FUNCTION_BLOCK "FB_MFC_Sort_COY_Result"
{ S7_Optimized_Access := 'TRUE' }
VERSION : 0.1
// ATTRIBUTES
// AUTO_NUMBER = True
// BLOCK_NUMBER = 117
// END_ATTRIBUTES
   VAR_INPUT
      ii_GINRangeStart { ExternalAccessible := 'False'; ExternalVisible := 'False'; ExternalWritable := 'False'} : Int := 0;   // GIN range start value
      ii_GINRangeEnd { ExternalAccessible := 'False'; ExternalVisible := 'False'; ExternalWritable := 'False'} : Int := 0;   // GIN range end value
      is_ObjectID : String[10];   // Recived parcel identifier
      ii_SourceNode : Int;   // ID Source Node
      ii_DestinationNode : Int;   // ID Destination Node
   END_VAR

   VAR_OUTPUT
      qx_Error : Bool;   // TRUE when collective block error occurred
      qx_Warning : Bool;   // TRUE when collective block warning occurred
   END_VAR

   VAR_IN_OUT
      iq_UDT_FifoHeader : "UDT_FifoHeader";   // FIFO header
      iqa_FifoData : Array[*] of "UDT_MessageV2";   // FIFO data buffer
      iqi_MessageSequenceNumber : Int;   // Message number
   END_VAR

   VAR
      ss_FB_HeartbeatPulse : "FB_Pulse";   // Heartbeat send pulse generator
      s_UDT_MessageArray : "UDT_MessageV2";   // Message array byte
      s_UDT_MessageHeader : "UDT_MFCSortMessageHeader";   // Message header
      ss_MessageBody : Struct   // Message body
         MsgID : Word;   // Message ID
         MsgLength : Word;   // Message length
         VID : Array[1..16] of Byte;   // Virtual Item Identifier
         PieceID : Array[1..40] of Byte;   // Piece ID
         Group : Byte;   // Group
         Level : Byte;   // Level
         Result : Byte;   // Result
         Eom : Byte;   // End of message
      END_STRUCT;
      ss_MessageData : Struct   // Message data
         VID : Array[1..16] of Byte;   // Virtual Item Identifier
         PieceID : Array[1..40] of Byte;   // Piece ID
         Group : String[1];   // Group
         Level : String[1];   // Level
         Result : String[1];   // Result
      END_STRUCT;
      ss_Status : Struct   // Status structure
         FIFOStatus : "UDT_FifoStatus";
         FIFOError { S7_SetPoint := 'True'} : Bool;   //  FIFO error
         FIFOWarning { S7_SetPoint := 'True'} : Bool;   // FIFO warning
         InvalidMessageArraySize : Bool;   // Message array is too short for message
         InvalidTimeInterval : Bool;   // Heartbeat time interval lower than zero
      END_STRUCT;
      sS_Old_Object_ID : String[10];   // Value from previous PLC cycle
      sdi_SerializePosition : DInt;   // Position in array where serialize finished writing data +1
      si_MaximumMessageLength : Int;   // Maximum number of elements in message array
      si_SerializeStatus : Int;   // Function serialize status
      sx_NewData : Bool;   // True - send a message to the MFC
   END_VAR

   VAR_TEMP
      ti_Loop_GIN : Int;   // Loop counter for DB_GIN
      ti_Loop : Int;   // Loop counter
   END_VAR

   VAR CONSTANT
      ci_MessageLength : Word := 16#003F;   // 10#0063 = 16#003F - Message length
      ci_MsgID : Word := 16#0137;   // 10#0311 = 16#0137 - Message ID
      ci_MsgLength : Word := 16#003B;   // 10#0059 = 16#003B - Message length
      ci_Som : Byte := 16#FD;   // Start of message
      ci_Eom : Byte := 16#FE;   // End of message
   END_VAR


BEGIN
	(*
	----------------------------------------------------------------------------------------
	|                                                                                      |
	|  Copyright  2023             FORTNA Europe BV                                        |
	|  All Rights Reserved         Netherlands                                             |
	|                                                                                      |
	----------------------------------------------------------------------------------------
	Version history:
	Date        | Version   | Author       | Remark
	----------------------------------------------------------------------------------------
	24/04/2023  | 1.0       | S. Nikodem   | Release TIA 17 | DHL Munich 2023
	03/10/2023  | 1.1       | S. Nikodem   | Update
	13/03/2023  | 1.2       | S. Nieswiec  | Updated for new Baseline
	02/05/2024  | 1.3       | J.Majer      | Datatype conversions changed from automatic to explicit, to accomodate IEC 61131-3 standard
	*)

	REGION 1 – FIFO header status update

	    // Mode 'S' - FIFO register status update.
	    "FC_Fifo"(ic_Mode := 'S',
	              qUDT_Status => #ss_Status.FIFOStatus,
	              qx_Error => #ss_Status.FIFOError,
	              qx_Warning => #ss_Status.FIFOWarning,
	              iqv_Data := #s_UDT_MessageArray,
	              iqUDT_FifoHeader := #iq_UDT_FifoHeader,
	              iqv_DataBuffer := #iqa_FifoData);

	END_REGION

	REGION 2 – Data preparation

	    //Generation message when is new parcel
	    #sx_NewData := (#is_ObjectID <> #sS_Old_Object_ID) AND NOT (#is_ObjectID = '');
	    // Save last value
	    #sS_Old_Object_ID := #is_ObjectID;

	    IF #sx_NewData THEN

	        FOR #ti_Loop_GIN := #ii_GINRangeStart TO #ii_GINRangeEnd DO

	            IF "DB_GIN".GIN[#ti_Loop_GIN].DHL.ObjectID = #is_ObjectID THEN

	                //VID
	                FOR #ti_Loop := 1 TO 16 DO

	                    #ss_MessageData.VID[#ti_Loop] := CHAR_TO_BYTE("DB_GIN".GIN[#ti_Loop_GIN].DHL.VID[#ti_Loop]);

	                END_FOR;

	                //Piece ID
	                FOR #ti_Loop := 1 TO 40 DO

	                    #ss_MessageData.PieceID[#ti_Loop] := CHAR_TO_BYTE("DB_GIN".GIN[#ti_Loop_GIN].DHL.PieceID[#ti_Loop]);

	                END_FOR;

	                //Group
	                #ss_MessageData.Group := "DB_GIN".GIN[#ti_Loop_GIN].DHL.Xray.Group;

	                //Level
	                #ss_MessageData.Level := "DB_GIN".GIN[#ti_Loop_GIN].DHL.Xray.Level;

	                //Result
	                #ss_MessageData.Result := "DB_GIN".GIN[#ti_Loop_GIN].DHL.Xray.Result;

	            END_IF;

	        END_FOR;

	    END_IF;

	END_REGION

	REGION 3 – Message array size validation

	    // Get size of the array.
	    #si_MaximumMessageLength := "FC_GetNrOfArrayEl"(#s_UDT_MessageArray.Bytes);

	    // Message array size validation.
	    #ss_Status.InvalidMessageArraySize := WORD_TO_INT(#ci_MessageLength) > #si_MaximumMessageLength;

	END_REGION


	REGION 4 – Message preparation

	    // FIFO full check.
	    IF NOT #iq_UDT_FifoHeader.Status.Full
	    THEN
	        // Errors and send pulse check.
	        IF NOT #ss_Status.FIFOError
	            AND NOT #ss_Status.InvalidMessageArraySize
	            AND #sx_NewData
	        THEN

	            REGION 4.1 – Header preparation

	                // Check sequence number. If it is equal or greater than 255 reset it to 1.
	                IF #iqi_MessageSequenceNumber <= 255
	                THEN
	                    #iqi_MessageSequenceNumber += 1;
	                ELSE
	                    #iqi_MessageSequenceNumber := 1;
	                END_IF;

	                // Write parts of the header into structure.
	                #s_UDT_MessageHeader.SOM := #ci_Som;
	                #s_UDT_MessageHeader.SourceNode := INT_TO_BYTE(#ii_SourceNode);
	                #s_UDT_MessageHeader.DestinationNode := INT_TO_BYTE(#ii_DestinationNode);
	                #s_UDT_MessageHeader.SeqNumber := INT_TO_BYTE(#iqi_MessageSequenceNumber);
	                #s_UDT_MessageHeader.DataLength := #ci_MessageLength;
	                #s_UDT_MessageHeader.NumMsg := 1;

	                // Write parts of the body into structure.
	                #ss_MessageBody.MsgID := #ci_MsgID;
	                #ss_MessageBody.MsgLength := #ci_MsgLength;
	                #ss_MessageBody.VID := #ss_MessageData.VID;
	                #ss_MessageBody.PieceID := #ss_MessageData.PieceID;
	                #ss_MessageBody.Group := CHAR_TO_BYTE(STRING_TO_CHAR(#ss_MessageData.Group));
	                #ss_MessageBody.Level := CHAR_TO_BYTE(STRING_TO_CHAR(#ss_MessageData.Level));
	                #ss_MessageBody.Result := CHAR_TO_BYTE(STRING_TO_CHAR(#ss_MessageData.Result));
	                #ss_MessageBody.Eom := #ci_Eom;

	            END_REGION

	            REGION 4.2 – Convert message into array of bytes

	                // Initialize the header serialize position and convert header structure into array of bytes.
	                #sdi_SerializePosition := 0;
	                #si_SerializeStatus := Serialize(SRC_VARIABLE := #s_UDT_MessageHeader,
	                                                 DEST_ARRAY => #s_UDT_MessageArray.Bytes,
	                                                 POS := #sdi_SerializePosition);

	                // Initialize the body serialize position and convert header structure into array of bytes
	                #si_SerializeStatus := Serialize(SRC_VARIABLE := #ss_MessageBody,
	                                                 DEST_ARRAY => #s_UDT_MessageArray.Bytes,
	                                                 POS := #sdi_SerializePosition);

	            END_REGION

	            REGION 4.3 – Write message into the FIFO buffer

	                // Mode 'W' - Write FIFO record.
	                "FC_Fifo"(ic_Mode := 'W',
	                          qUDT_Status => #ss_Status.FIFOStatus,
	                          qx_Error => #ss_Status.FIFOError,
	                          qx_Warning => #ss_Status.FIFOWarning,
	                          iqv_Data := #s_UDT_MessageArray,
	                          iqUDT_FifoHeader := #iq_UDT_FifoHeader,
	                          iqv_DataBuffer := #iqa_FifoData);

	            END_REGION

	        END_IF;
	    ELSE
	        // If FIFO is full set FIFO main and FIFO full errors.
	        #ss_Status.FIFOError := TRUE;
	        #ss_Status.FIFOStatus.FifoFull := TRUE;
	    END_IF;

	END_REGION

	REGION 5 - Status

	    // Parametrization collective error output.
	    #qx_Error :=
	    #ss_Status.FIFOError
	    OR #ss_Status.InvalidTimeInterval
	    OR #ss_Status.InvalidMessageArraySize;

	    // Parametrization collective warning output.
	    #qx_Warning := #ss_Status.FIFOWarning;

	END_REGION
END_FUNCTION_BLOCK

TYPE "UDT_PECUpdateConfiguration"
TITLE = UDT_PECConfiguration
VERSION : 0.1
//User-defined structure of PEC parameters.
   STRUCT
      Distance : DInt;   // Distance between photo eye and the end of conveyor [mm]
      JamDisplacementLimit : Int;   // Limit displacement with PEC blocked o detect jam [cm]
      TimeOnDelay : UDInt;   // Photo eye time on delay [ms]
      TimeOffDelay : UDInt;   // Photo eye time off delay [ms]
      ParcelLengthFilter : Bool := TRUE;   // Parcel length filter
      ResetWithPECBlocked { ExternalAccessible := 'False'; ExternalVisible := 'False'; ExternalWritable := 'False'} : Bool;   // When 'True' Allow reset system after jam with PEC blocked
      SearchWindowFwd : Int;   // Search window in forward direction [cm]
      SearchWindowRvs : Int;   // Search window in reverse direction [cm]
      GINRangeStart : Int;   // GIN range start value
      GINRangeEnd : Int;   // GIN range end value
      NrOfTeachParcels : Int;   // Number of parcels to teach
      DefaultGIN : Int := 1;   // Default GIN record
      MaxLost : Int;   // Maximum number of lost parcels in a row
      GenerationPoint { ExternalAccessible := 'False'; ExternalVisible := 'False'; ExternalWritable := 'False'} : Bool;   // Generation point
      NegativeGINDelete { ExternalAccessible := 'False'; ExternalVisible := 'False'; ExternalWritable := 'False'} : Bool;   // True when negative GIN has to be deleted
      ParcelLengthMeasurement { ExternalAccessible := 'False'; ExternalVisible := 'False'; ExternalWritable := 'False'} : Bool;   // Parcel length measurement
      GapLengthMeasurement { ExternalAccessible := 'False'; ExternalVisible := 'False'; ExternalWritable := 'False'} : Bool;   // Gap length measurement
   END_STRUCT;

END_TYPE

FUNCTION_BLOCK "FB_MFC_Sort_COY_ReceiveResult"
{ S7_Optimized_Access := 'TRUE' }
VERSION : 0.1
// ATTRIBUTES
// AUTO_NUMBER = True
// BLOCK_NUMBER = 115
// END_ATTRIBUTES
   VAR_INPUT
      is_VID { ExternalAccessible := 'False'; ExternalVisible := 'False'; ExternalWritable := 'False'} : String[16];   // Virtual Item Identifier (VID)
      is_PieceID { ExternalAccessible := 'False'; ExternalVisible := 'False'; ExternalWritable := 'False'} : String[40];   // Piece ID barcodes
      is_Group { ExternalAccessible := 'False'; ExternalVisible := 'False'; ExternalWritable := 'False'} : String[1];   // The group field is used to identify the group of the operator decisions came from in a
      is_Level { ExternalAccessible := 'False'; ExternalVisible := 'False'; ExternalWritable := 'False'} : String[1];   // Level field is used to identify which level the operator decision came from in a
      is_Result { ExternalAccessible := 'False'; ExternalVisible := 'False'; ExternalWritable := 'False'} : String[1];   // Results can be indicated with the following
      ii_SourceNode { ExternalAccessible := 'False'; ExternalVisible := 'False'; ExternalWritable := 'False'} : Int;   // ID Source Node
      ii_DestinationNode { ExternalAccessible := 'False'; ExternalVisible := 'False'; ExternalWritable := 'False'} : Int;   // ID Destination Node
   END_VAR

   VAR_OUTPUT
      qx_Error { ExternalAccessible := 'False'; ExternalVisible := 'False'; ExternalWritable := 'False'} : Bool;   // TRUE when collective block error occurred
      qx_Warning { ExternalAccessible := 'False'; ExternalVisible := 'False'; ExternalWritable := 'False'} : Bool;   // TRUE when collective block warning occurred
   END_VAR

   VAR_IN_OUT
      iq_UDT_FifoHeader : "UDT_FifoHeader";   // FIFO header
      iqa_FifoData : Array[*] of "UDT_MessageV2";   // FIFO data buffer
      iqi_MessageSequenceNumber { ExternalAccessible := 'False'; ExternalVisible := 'False'; ExternalWritable := 'False'} : Int;   // Message number
   END_VAR

   VAR
      ss_FB_HeartbeatPulse { ExternalAccessible := 'False'; ExternalVisible := 'False'; ExternalWritable := 'False'; S7_SetPoint := 'False'} : "FB_Pulse";   // Heartbeat send pulse generator
      s_UDT_MessageArray { ExternalAccessible := 'False'; ExternalVisible := 'False'; ExternalWritable := 'False'; S7_SetPoint := 'False'} : "UDT_MessageV2";   // Message array byte
      s_UDT_MessageHeader { ExternalAccessible := 'False'; ExternalVisible := 'False'; ExternalWritable := 'False'; S7_SetPoint := 'False'} : "UDT_MFCSortMessageHeader";   // Message header
      ss_MessageBody { ExternalAccessible := 'False'; ExternalVisible := 'False'; ExternalWritable := 'False'} : Struct   // Message body
         MsgID { ExternalAccessible := 'False'; ExternalVisible := 'False'; ExternalWritable := 'False'} : Word;   // Message ID
         MsgLength { ExternalAccessible := 'False'; ExternalVisible := 'False'; ExternalWritable := 'False'} : Word;   // Message length
         VID { ExternalAccessible := 'False'; ExternalVisible := 'False'; ExternalWritable := 'False'} : Array[1..16] of Byte;   // Virtual Item Identifier
         PieceID { ExternalAccessible := 'False'; ExternalVisible := 'False'; ExternalWritable := 'False'} : Array[1..40] of Byte;   // Piece ID
         Group { ExternalAccessible := 'False'; ExternalVisible := 'False'; ExternalWritable := 'False'} : Byte;   // Group
         Level { ExternalAccessible := 'False'; ExternalVisible := 'False'; ExternalWritable := 'False'} : Byte;   // Level
         Result { ExternalAccessible := 'False'; ExternalVisible := 'False'; ExternalWritable := 'False'} : Byte;   // Result
         Eom { ExternalAccessible := 'False'; ExternalVisible := 'False'; ExternalWritable := 'False'} : Byte;   // End of message
      END_STRUCT;
      ss_MessageData { ExternalAccessible := 'False'; ExternalVisible := 'False'; ExternalWritable := 'False'} : Struct   // Message data
         VID { ExternalAccessible := 'False'; ExternalVisible := 'False'; ExternalWritable := 'False'} : Array[1..16] of Byte;   // Virtual Item Identifier
         PieceID { ExternalAccessible := 'False'; ExternalVisible := 'False'; ExternalWritable := 'False'} : Array[1..40] of Byte;   // Piece ID
         Group { ExternalAccessible := 'False'; ExternalVisible := 'False'; ExternalWritable := 'False'} : String[1];   // Group
         Level { ExternalAccessible := 'False'; ExternalVisible := 'False'; ExternalWritable := 'False'} : String[1];   // Level
         Result { ExternalAccessible := 'False'; ExternalVisible := 'False'; ExternalWritable := 'False'} : String[1];   // Result
      END_STRUCT;
      ss_Status { ExternalAccessible := 'False'; ExternalVisible := 'False'; ExternalWritable := 'False'} : Struct   // Status structure
         FIFOStatus { ExternalAccessible := 'False'; ExternalVisible := 'False'; ExternalWritable := 'False'} : "UDT_FifoStatus";
         FIFOError { ExternalAccessible := 'False'; ExternalVisible := 'False'; ExternalWritable := 'False'; S7_SetPoint := 'True'} : Bool;   //  FIFO error
         FIFOWarning { ExternalAccessible := 'False'; ExternalVisible := 'False'; ExternalWritable := 'False'; S7_SetPoint := 'True'} : Bool;   // FIFO warning
         InvalidMessageArraySize { ExternalAccessible := 'False'; ExternalVisible := 'False'; ExternalWritable := 'False'} : Bool;   // Message array is too short for message
         InvalidTimeInterval { ExternalAccessible := 'False'; ExternalVisible := 'False'; ExternalWritable := 'False'} : Bool;   // Heartbeat time interval lower than zero
      END_STRUCT;
      sdi_SerializePosition { ExternalAccessible := 'False'; ExternalVisible := 'False'; ExternalWritable := 'False'} : DInt;   // Position in array where serialize finished writing data +1
      si_MaximumMessageLength { ExternalAccessible := 'False'; ExternalVisible := 'False'; ExternalWritable := 'False'} : Int;   // Maximum number of elements in message array
      si_SerializeStatus { ExternalAccessible := 'False'; ExternalVisible := 'False'; ExternalWritable := 'False'} : Int;   // Function serialize status
      sx_NewData { ExternalAccessible := 'False'; ExternalVisible := 'False'; ExternalWritable := 'False'} : Bool;   // New data received
      ss_PieceIDOld { ExternalAccessible := 'False'; ExternalVisible := 'False'; ExternalWritable := 'False'} : String[40];   // Piece ID barcodes old value
   END_VAR

   VAR_TEMP
      ti_Loop : Int;
   END_VAR

   VAR CONSTANT
      ci_MessageLength : Word := 16#003F;   // 10#0063 = 16#003F - Message length
      ci_MsgID : Word := 16#0137;   // 10#0311 = 16#0137 - Message ID
      ci_MsgLength : Word := 16#003B;   // 10#0059 = 16#003B - Message length
      ci_Som : Byte := 16#FD;   // Start of message
      ci_Eom : Byte := 16#FE;   // End of message
   END_VAR


BEGIN
	(*
	----------------------------------------------------------------------------------------
	|                                                                                      |
	|  Copyright  2023             FORTNA Europe BV                                        |
	|  All Rights Reserved         Netherlands                                             |
	|                                                                                      |
	----------------------------------------------------------------------------------------
	Version history:
	Date        | Version   | Author       | Remark
	----------------------------------------------------------------------------------------
	05/10/2023  | 1.0       | S. Nikodem   | Release TIA 17 | DHL Munich 2023
	13/03/2023  | 1.1       | S. Nieswiec  | Updated for new Baseline
	02/05/2024  | 1.2       | J.Majer      | Datatype conversions changed from automatic to explicit, to accomodate IEC 61131-3 standard
	*)

	REGION 1 – FIFO header status update

	    // Mode 'S' - FIFO register status update.
	    "FC_Fifo"(ic_Mode := 'S',
	              qUDT_Status => #ss_Status.FIFOStatus,
	              qx_Error => #ss_Status.FIFOError,
	              qx_Warning => #ss_Status.FIFOWarning,
	              iqv_Data := #s_UDT_MessageArray,
	              iqUDT_FifoHeader := #iq_UDT_FifoHeader,
	              iqv_DataBuffer := #iqa_FifoData);

	END_REGION

	REGION 2 – Data preparation

	    IF #is_PieceID <> #ss_PieceIDOld AND NOT (#ss_PieceIDOld = '') THEN

	        //Save
	        #ss_PieceIDOld := #is_PieceID;

	        //VID
	        FOR #ti_Loop := 1 TO 16 DO

	            #ss_MessageData.VID[#ti_Loop] := CHAR_TO_BYTE(#is_VID[#ti_Loop]);

	        END_FOR;

	        //Piece ID
	        FOR #ti_Loop := 1 TO 40 DO

	            #ss_MessageData.PieceID[#ti_Loop] := CHAR_TO_BYTE(#is_PieceID[#ti_Loop]);

	        END_FOR;

	        //Group
	        #ss_MessageData.Group := #is_Group;

	        //Level
	        #ss_MessageData.Level := #is_Level;

	        //Result
	        #ss_MessageData.Result := #is_Result;

	        //New data received
	        #sx_NewData := TRUE;

	    END_IF;


	END_REGION

	REGION 3 – Message array size validation

	    // Get size of the array.
	    #si_MaximumMessageLength := "FC_GetNrOfArrayEl"(#s_UDT_MessageArray.Bytes);

	    // Message array size validation.
	    #ss_Status.InvalidMessageArraySize := WORD_TO_INT(#ci_MessageLength) > #si_MaximumMessageLength;

	END_REGION


	REGION 4 – Message preparation

	    // FIFO full check.
	    IF NOT #iq_UDT_FifoHeader.Status.Full
	    THEN
	        // Errors and send pulse check.
	        IF NOT #ss_Status.FIFOError
	            AND NOT #ss_Status.InvalidMessageArraySize
	            AND #sx_NewData
	        THEN

	            REGION 4.1 – Header preparation

	                // Check sequence number. If it is equal or greater than 255 reset it to 1.
	                IF #iqi_MessageSequenceNumber <= 255
	                THEN
	                    #iqi_MessageSequenceNumber += 1;
	                ELSE
	                    #iqi_MessageSequenceNumber := 1;
	                END_IF;

	                // Write parts of the header into structure.
	                #s_UDT_MessageHeader.SOM := #ci_Som;
	                #s_UDT_MessageHeader.SourceNode := INT_TO_BYTE(#ii_SourceNode);
	                #s_UDT_MessageHeader.DestinationNode := INT_TO_BYTE(#ii_DestinationNode);
	                #s_UDT_MessageHeader.SeqNumber := INT_TO_BYTE(#iqi_MessageSequenceNumber);
	                #s_UDT_MessageHeader.DataLength := #ci_MessageLength;
	                #s_UDT_MessageHeader.NumMsg := 1;

	                // Write parts of the body into structure.
	                #ss_MessageBody.MsgID := #ci_MsgID;
	                #ss_MessageBody.MsgLength := #ci_MsgLength;
	                #ss_MessageBody.VID := #ss_MessageData.VID;
	                #ss_MessageBody.PieceID := #ss_MessageData.PieceID;
	                #ss_MessageBody.Group := CHAR_TO_BYTE(STRING_TO_CHAR(#ss_MessageData.Group));
	                #ss_MessageBody.Level := CHAR_TO_BYTE(STRING_TO_CHAR(#ss_MessageData.Level));
	                #ss_MessageBody.Result := CHAR_TO_BYTE(STRING_TO_CHAR(#ss_MessageData.Result));
	                #ss_MessageBody.Eom := #ci_Eom;

	            END_REGION

	            REGION 4.2 – Convert message into array of bytes

	                // Initialize the header serialize position and convert header structure into array of bytes.
	                #sdi_SerializePosition := 0;
	                #si_SerializeStatus := Serialize(SRC_VARIABLE := #s_UDT_MessageHeader,
	                                                 DEST_ARRAY => #s_UDT_MessageArray.Bytes,
	                                                 POS := #sdi_SerializePosition);

	                // Initialize the body serialize position and convert header structure into array of bytes
	                #si_SerializeStatus := Serialize(SRC_VARIABLE := #ss_MessageBody,
	                                                 DEST_ARRAY => #s_UDT_MessageArray.Bytes,
	                                                 POS := #sdi_SerializePosition);

	            END_REGION

	            REGION 4.3 – Write message into the FIFO buffer

	                // Mode 'W' - Write FIFO record.
	                "FC_Fifo"(ic_Mode := 'W',
	                          qUDT_Status => #ss_Status.FIFOStatus,
	                          qx_Error => #ss_Status.FIFOError,
	                          qx_Warning => #ss_Status.FIFOWarning,
	                          iqv_Data := #s_UDT_MessageArray,
	                          iqUDT_FifoHeader := #iq_UDT_FifoHeader,
	                          iqv_DataBuffer := #iqa_FifoData);

	            END_REGION

	            //Reset
	            #sx_NewData := False;

	        END_IF;
	    ELSE
	        // If FIFO is full set FIFO main and FIFO full errors.
	        #ss_Status.FIFOError := TRUE;
	        #ss_Status.FIFOStatus.FifoFull := TRUE;
	    END_IF;

	END_REGION

	REGION 5 - Status

	    // Parametrization collective error output.
	    #qx_Error :=
	    #ss_Status.FIFOError
	    OR #ss_Status.InvalidTimeInterval
	    OR #ss_Status.InvalidMessageArraySize;

	    // Parametrization collective warning output.
	    #qx_Warning := #ss_Status.FIFOWarning;

	END_REGION
END_FUNCTION_BLOCK

TYPE "UDT_XrayRapiscanConfiguration"
VERSION : 0.1
   STRUCT
      EstopResetPluse : UDInt;   // Time how long the pulse should be active [ms]
      IDmessageTimeout : UDInt;   // The maximum time after which Xray must receive a Bag ID [ms]
      BagIDPoint : UDInt;   // Place in the Xray conveyor tracking from which Bag ID is to be taken [cm]
      ScanningWindowStartPoint : Int;   // Scanning window a start point in the Xray conveyor tracking [cm]
      ScanningWindowEndPoint : Int;   // Scanning window a end point in the Xray conveyor tracking [cm]
      BackBeltDistance : UDInt;   // Back belt distance [cm]
      XrayConveyor { S7_SetPoint := 'False'} : "UDT_ConveyorCommonConfiguration";   // Conveyor configuration
      SerialCommunicationConfiguration { S7_SetPoint := 'False'} : "UDT_SerialComConfiguration";
   END_STRUCT;

END_TYPE

TYPE "UDT_RapiscanStatus"
TITLE = UDT_HS10080XCTStatus
VERSION : 0.1
//User-defined structure of FB_Xray_HS10080XCT function block status.
   STRUCT
      Status : Int;   // Status number
      XraySpecific : Struct   // Equipment specific warnings and errors
         XrayEnergised : Bool;   // Xray Energised
         XrayFault : Bool;   // Xray Fault
         XrayRdyRCV : Bool;   // Xray Ready receive
         XrayRdySend : Bool;   // Xray Ready send
         BagScanning : Bool;   // Xray bag scaning
         TransportMode : Bool;   // Transport mode active
         BackBelt : Bool;   // Backbelt functinality active
      END_STRUCT;
      ConvSpecific : Struct   // Equipment specific warnings and errors
         Status : Int;   // Status number
         Conv_ERR : Bool;   // Conveyor is in error
         Encoder_ERR : Bool;   // Encoder error
         ConvRunFWD : Bool;   // Conveyor run forward direction
         ConvRunREV : Bool;   // Conveyor run reverse direction
      END_STRUCT;
   END_STRUCT;

END_TYPE

TYPE "UDT_RapiscanStatistics"
TITLE = UDT_HS10080XCTStatistics
VERSION : 0.1
//User-defined structure of FB_Xray_HS10080XCT function block statistics.
   STRUCT
      TransportMode : "UDT_EventStatistic";   // Running in transit mode
      EncoderError : "UDT_EventStatistic";   // One of the encoders has faulted
   END_STRUCT;

END_TYPE

FUNCTION_BLOCK "FB_VFD_FishBone"
{ S7_Optimized_Access := 'TRUE' }
VERSION : 0.1
// ATTRIBUTES
// AUTO_NUMBER = True
// BLOCK_NUMBER = 245
// END_ATTRIBUTES
   VAR_INPUT
      i_UDT_MultiControlConfiguration { ExternalAccessible := 'False'; ExternalVisible := 'False'; ExternalWritable := 'False'} : "UDT_VFD_MultiControl_Configuration";   //   VFD configuration structure
      i_UDT_MultiControl_1_Inputs { ExternalAccessible := 'False'; ExternalVisible := 'False'; ExternalWritable := 'False'} : "UDT_VFD_MultiControl_PI";   //   VFD inputs structure
      i_UDT_MultiControl_2_Inputs { ExternalAccessible := 'False'; ExternalVisible := 'False'; ExternalWritable := 'False'} : "UDT_VFD_MultiControl_PI";   //   VFD inputs structure
      is_MultiControl_1_PNDeviceName { ExternalAccessible := 'False'; ExternalVisible := 'False'; ExternalWritable := 'False'} : String;   // MultiControl 1 Profinet device name
      is_MultiControl_2_PNDeviceName { ExternalAccessible := 'False'; ExternalVisible := 'False'; ExternalWritable := 'False'} : String;   // MultiControl 2 Profinet device name
      ix_PowerOK { ExternalAccessible := 'False'; ExternalVisible := 'False'; ExternalWritable := 'False'} : Bool;   //   TRUE when External Power OK
      ix_SafetyOK { ExternalAccessible := 'False'; ExternalVisible := 'False'; ExternalWritable := 'False'} : Bool;   //   TRUE when Safety OK
   END_VAR

   VAR_OUTPUT
      q_UDT_HMIStatus { ExternalAccessible := 'False'; ExternalVisible := 'False'; ExternalWritable := 'False'} : "UDT_VfdStatus";   //   HMI status structure
      qsi_VFDSpeed { ExternalAccessible := 'False'; ExternalVisible := 'False'; ExternalWritable := 'False'} : SInt;   //   VFD speed setpoint
   END_VAR

   VAR_IN_OUT
      iq_UDT_ConveyorInterface : "UDT_ConveyorInterface";   //   Conveyor interface structure
      iq_UDT_VFDStatistics : "UDT_VfdStatistics";   //   Statistics structure
      iq_UDT_Equipment : "UDT_EquipmentControl";   // equipment control commands
   END_VAR

   VAR
      s_FB_VFD_MultiControl_1 { ExternalAccessible := 'False'; ExternalVisible := 'False'; ExternalWritable := 'False'; S7_SetPoint := 'False'} : "FB_VFD_MultiControl_V4";   // FB multi control 1
      s_FB_VFD_MultiControl_2 { ExternalAccessible := 'False'; ExternalVisible := 'False'; ExternalWritable := 'False'; S7_SetPoint := 'False'} : "FB_VFD_MultiControl_V4";   // FB multi control 2
      s_UDT_MultiControlConfiguration { ExternalAccessible := 'False'; ExternalVisible := 'False'; ExternalWritable := 'False'; S7_SetPoint := 'False'} : "UDT_VFD_MultiControl_Configuration";   //   VFD configuration structure
      s_UDT_Multicontrol_1_HMIStatus { ExternalAccessible := 'False'; ExternalVisible := 'False'; ExternalWritable := 'False'; S7_SetPoint := 'False'} : "UDT_VfdStatus";   //   HMI status structure
      s_UDT_Multicontrol_2_HMIStatus { ExternalAccessible := 'False'; ExternalVisible := 'False'; ExternalWritable := 'False'; S7_SetPoint := 'False'} : "UDT_VfdStatus";   //   HMI status structure
      s_UDT_Multicontrol_1_Statistics { ExternalAccessible := 'False'; ExternalVisible := 'False'; ExternalWritable := 'False'; S7_SetPoint := 'False'} : "UDT_VfdStatistics";   //   Statistics structure
      s_UDT_Multicontrol_2_Statistics { ExternalAccessible := 'False'; ExternalVisible := 'False'; ExternalWritable := 'False'; S7_SetPoint := 'False'} : "UDT_VfdStatistics";   //   Statistics structure
   END_VAR


BEGIN
	(*
	----------------------------------------------------------------------------------------
	|                                                                                      |
	|  Copyright  2023             FORTNA Europe BV                                        |
	|  All Rights Reserved         Netherlands                                             |
	|                                                                                      |
	----------------------------------------------------------------------------------------

	Version history:
	Date        | Version   | Author        | Remark
	----------------------------------------------------------------------------------------
	08/12/2022  | 1.0       | S. Nikodem    | Initial version | DHL Munich 2023
	13/03/2024  | 1.1       | S. Nieswiec       | Added to new baseline
	*)

	REGION 1 - MultiControl 1

	    //Copy configuration to static memory
	    #s_UDT_MultiControlConfiguration := #i_UDT_MultiControlConfiguration;

	    //Write Profinet name
	    #s_UDT_MultiControlConfiguration.VFDPNDeviceName := #is_MultiControl_1_PNDeviceName;

	    //Call MultiControl function for 4 motors handling
	    #s_FB_VFD_MultiControl_1(i_UDT_VFDConfiguration := #i_UDT_MultiControlConfiguration,
	                             i_UDT_VFDInputs := #i_UDT_MultiControl_1_Inputs,
	                             ix_PowerOK := #ix_PowerOK,
	                             ix_SafetyOK := #ix_SafetyOK,
	                             q_UDT_HMIStatus => #q_UDT_HMIStatus,
	                             qsi_UDT_VFDSpeed => #qsi_VFDSpeed,
	                             iq_UDT_ConveyorInterface := #iq_UDT_ConveyorInterface,
	                             iq_UDT_VFDStatistics := #iq_UDT_VFDStatistics,
	                             iq_UDT_Equipment := #iq_UDT_Equipment);

	END_REGION

	REGION 2 - MultiControl 2

	    //Write Profinet name
	    #s_UDT_MultiControlConfiguration.VFDPNDeviceName := #is_MultiControl_2_PNDeviceName;

	    //Call MultiControl function for 4 motors handling
	    #s_FB_VFD_MultiControl_2(i_UDT_VFDConfiguration := #i_UDT_MultiControlConfiguration,
	                             i_UDT_VFDInputs := #i_UDT_MultiControl_2_Inputs,
	                             ix_PowerOK := #ix_PowerOK,
	                             ix_SafetyOK := #ix_SafetyOK,
	                             q_UDT_HMIStatus => #q_UDT_HMIStatus,
	                             qsi_UDT_VFDSpeed => #qsi_VFDSpeed,
	                             iq_UDT_ConveyorInterface := #iq_UDT_ConveyorInterface,
	                             iq_UDT_VFDStatistics := #iq_UDT_VFDStatistics,
	                             iq_UDT_Equipment := #iq_UDT_Equipment);

	END_REGION

	REGION 3 - HMI Status

	    #q_UDT_HMIStatus.PNSlaveNotonline := #s_UDT_Multicontrol_1_HMIStatus.PNSlaveNotonline OR #s_UDT_Multicontrol_2_HMIStatus.PNSlaveNotonline;
	    #q_UDT_HMIStatus.PNSlaveError := #s_UDT_Multicontrol_1_HMIStatus.PNSlaveError OR #s_UDT_Multicontrol_2_HMIStatus.PNSlaveError;
	    #q_UDT_HMIStatus.InternalError := #s_UDT_Multicontrol_1_HMIStatus.InternalError OR #s_UDT_Multicontrol_2_HMIStatus.InternalError;

	END_REGION

	REGION 4- Statistics

	    //Piority for first MultiControl

	    //PNSlaveNotOnline
	    #iq_UDT_VFDStatistics.PNSlaveNotOnline.LastEventSeconds := #s_UDT_Multicontrol_1_Statistics.PNSlaveNotOnline.LastEventSeconds;
	    #iq_UDT_VFDStatistics.PNSlaveNotOnline.NumberOfTimes := #s_UDT_Multicontrol_1_Statistics.PNSlaveNotOnline.NumberOfTimes + #s_UDT_Multicontrol_2_Statistics.PNSlaveNotOnline.NumberOfTimes;
	    #iq_UDT_VFDStatistics.PNSlaveNotOnline.TotalEventSeconds := #s_UDT_Multicontrol_1_Statistics.PNSlaveNotOnline.TotalEventSeconds + #s_UDT_Multicontrol_2_Statistics.PNSlaveNotOnline.TotalEventSeconds;

	    //PNSlaveError
	    #iq_UDT_VFDStatistics.PNSlaveError.LastEventSeconds := #s_UDT_Multicontrol_1_Statistics.PNSlaveError.LastEventSeconds;
	    #iq_UDT_VFDStatistics.PNSlaveError.NumberOfTimes := #s_UDT_Multicontrol_1_Statistics.PNSlaveError.NumberOfTimes + #s_UDT_Multicontrol_2_Statistics.PNSlaveError.NumberOfTimes;
	    #iq_UDT_VFDStatistics.PNSlaveError.TotalEventSeconds := #s_UDT_Multicontrol_1_Statistics.PNSlaveError.TotalEventSeconds + #s_UDT_Multicontrol_2_Statistics.PNSlaveError.TotalEventSeconds;

	    //VFDInternalError
	    #iq_UDT_VFDStatistics.VFDInternalError.LastEventSeconds := #s_UDT_Multicontrol_1_Statistics.VFDInternalError.LastEventSeconds;
	    #iq_UDT_VFDStatistics.VFDInternalError.NumberOfTimes := #s_UDT_Multicontrol_1_Statistics.VFDInternalError.NumberOfTimes + #s_UDT_Multicontrol_2_Statistics.VFDInternalError.NumberOfTimes;
	    #iq_UDT_VFDStatistics.VFDInternalError.TotalEventSeconds := #s_UDT_Multicontrol_1_Statistics.VFDInternalError.TotalEventSeconds + #s_UDT_Multicontrol_2_Statistics.VFDInternalError.TotalEventSeconds;

	    //Running
	    //Piority for first MultiControl
	    #iq_UDT_VFDStatistics.Running := #s_UDT_Multicontrol_1_Statistics.Running;

	END_REGION



END_FUNCTION_BLOCK

FUNCTION_BLOCK "FB_ConveyorV2"
TITLE = FB_Conveyor_BiDirectional
{ S7_Optimized_Access := 'TRUE' }
AUTHOR : MHSE
FAMILY : Equimpent
VERSION : 3.0
// ATTRIBUTES
// AUTO_NUMBER = True
// BLOCK_NUMBER = 94
// END_ATTRIBUTES
//Function block to control the bi-directional conveyor.
   VAR_INPUT
      i_UDT_ConveyorConfiguration { ExternalAccessible := 'False'; ExternalVisible := 'False'; ExternalWritable := 'False'} : "UDT_ConveyorConfiguration";   //           Conveyor configuration structure
      idi_PEC_EoSDistance { ExternalAccessible := 'False'; ExternalVisible := 'False'; ExternalWritable := 'False'} : DInt;   //           Distance between photo eye and the end of conveyor [mm] in forward direction
      idi_PEC_BoSDistance { ExternalAccessible := 'False'; ExternalVisible := 'False'; ExternalWritable := 'False'} : DInt;   //           Distance between photo eye and the end of conveyor [mm] in reverse direction
      ii_ExternalSpeed { ExternalAccessible := 'False'; ExternalVisible := 'False'; ExternalWritable := 'False'} : Int;   //           External speed [mm/s]
      ix_SafetyOk { ExternalAccessible := 'False'; ExternalVisible := 'False'; ExternalWritable := 'False'} : Bool;   //           TRUE when safety is ok
      ix_24vOk { ExternalAccessible := 'False'; ExternalVisible := 'False'; ExternalWritable := 'False'} : Bool;   //           TRUE when 24VDC is healthy
      ix_400vOk { ExternalAccessible := 'False'; ExternalVisible := 'False'; ExternalWritable := 'False'} : Bool;   //           TRUE when 400VAC is healthy
      ix_HardwareOk { ExternalAccessible := 'False'; ExternalVisible := 'False'; ExternalWritable := 'False'} : Bool;   //           TRUE when  hardware is Ok
      ix_PEC_EoS { ExternalAccessible := 'False'; ExternalVisible := 'False'; ExternalWritable := 'False'} : Bool := TRUE;   //           TRUE when the end of section photoeye in forward direction is not blocked
      ix_PEC_BoS { ExternalAccessible := 'False'; ExternalVisible := 'False'; ExternalWritable := 'False'} : Bool := TRUE;   //           TRUE when the end of section photoeye in reverse direction is not blocked
      ix_ReverseDirection { ExternalAccessible := 'False'; ExternalVisible := 'False'; ExternalWritable := 'False'} : Bool;   //           FALSE when to run in forward direction and True to run in Reverse direction
      ix_ExternalRequestDieBack { ExternalAccessible := 'False'; ExternalVisible := 'False'; ExternalWritable := 'False'} : Bool;   //           External input to request die back
      ix_ExternalRequestHold { ExternalAccessible := 'False'; ExternalVisible := 'False'; ExternalWritable := 'False'} : Bool;   //           External input to request conveyor hold
      ix_ResetEnergySave { ExternalAccessible := 'False'; ExternalVisible := 'False'; ExternalWritable := 'False'} : Bool;   //           Reset energy save mode timer
   END_VAR

   VAR_OUTPUT
      q_UDT_HMIStatus { ExternalAccessible := 'False'; ExternalVisible := 'False'; ExternalWritable := 'False'} : "UDT_ConveyorStatus";   //           HMI status structure
      q_UDT_Status { ExternalAccessible := 'False'; ExternalVisible := 'False'; ExternalWritable := 'False'} : "UDT_CommonStatus";   //           Common status structure
   END_VAR

   VAR_IN_OUT
      iq_UDT_EquipmentControl : "UDT_EquipmentControl";   //           Equipment control structure
      iq_UDT_ConveyorCommand : "UDT_ConveyorCommand";   //           Conveyor command stucture
      iq_UDT_ConveyorInterface : "UDT_ConveyorInterface";   //           Interface structure
      iq_UDT_HandShakeUp : "UDT_ConveyorHandshake";   //           Upstream handshake structure in forward direction
      iq_UDT_HandShake : "UDT_ConveyorHandshake";   //           Handshake structure in forward direction
      iq_UDT_Statistics : "UDT_ConveyorStatistics";   //           Statistics structure
   END_VAR

   VAR
      s_UDT_CommonStatus { ExternalAccessible := 'False'; ExternalVisible := 'False'; ExternalWritable := 'False'; S7_SetPoint := 'False'} : "UDT_CommonStatus";   //           Common status structure
      s_UDT_CommonStatusOld { ExternalAccessible := 'False'; ExternalVisible := 'False'; ExternalWritable := 'False'; S7_SetPoint := 'False'} : "UDT_CommonStatus";   //           Auxiliary status structure
      s_UDT_HMIStatus { ExternalAccessible := 'False'; ExternalVisible := 'False'; ExternalWritable := 'False'; S7_SetPoint := 'False'} : "UDT_ConveyorStatus";   //           HMI status structure
      s_FB_CascadeModeTimer { ExternalAccessible := 'False'; ExternalVisible := 'False'; ExternalWritable := 'False'; S7_SetPoint := 'False'} : "FB_TimerOnOffDelay";   //           Timer to cascade start
      sdi_GapHeadToHeadConfiguration_Fwd { ExternalAccessible := 'False'; ExternalVisible := 'False'; ExternalWritable := 'False'} : DInt;   //           Preset forward gap head to head with correction [cm]
      sdi_GapTailToHeadConfiguration_Fwd { ExternalAccessible := 'False'; ExternalVisible := 'False'; ExternalWritable := 'False'} : DInt;   //           Preset forward gap tail to head with correction [cm]
      sdi_GapHeadToHeadConfiguration_Rvs { ExternalAccessible := 'False'; ExternalVisible := 'False'; ExternalWritable := 'False'} : DInt;   //           Preset reverse gap head to head with correction [cm]
      sdi_GapTailToHeadConfiguration_Rvs { ExternalAccessible := 'False'; ExternalVisible := 'False'; ExternalWritable := 'False'} : DInt;   //           Preset reverse gap tail to head with correction [cm]
   END_VAR
   VAR RETAIN
      sdi_AuxGapHeadToHeadCounter_Fwd { ExternalAccessible := 'False'; ExternalVisible := 'False'; ExternalWritable := 'False'} : DInt;   //           Aux variable to count the head to head
      sdi_AuxGapTailtoHeadCounter_Fwd { ExternalAccessible := 'False'; ExternalVisible := 'False'; ExternalWritable := 'False'} : DInt;   //           Aux variable to count the gap
      sdi_AuxGapHeadToHeadCounter_Rvs { ExternalAccessible := 'False'; ExternalVisible := 'False'; ExternalWritable := 'False'} : DInt;   //           Aux variable to count the head to head
      sdi_AuxGapTailtoHeadCounter_Rvs { ExternalAccessible := 'False'; ExternalVisible := 'False'; ExternalWritable := 'False'} : DInt;   //           Aux variable to count the gap
      sdi_Gap_Fwd { ExternalAccessible := 'False'; ExternalVisible := 'False'; ExternalWritable := 'False'} : DInt;   //           Gap between two products
      sdi_GapHeadToHead_Fwd { ExternalAccessible := 'False'; ExternalVisible := 'False'; ExternalWritable := 'False'} : DInt;   //           Head to head between two products
      sdi_Gap_Rvs { ExternalAccessible := 'False'; ExternalVisible := 'False'; ExternalWritable := 'False'} : DInt;   //           Gap between two products
      sdi_GapHeadToHead_Rvs { ExternalAccessible := 'False'; ExternalVisible := 'False'; ExternalWritable := 'False'} : DInt;   //           Head to head between two products
      sdi_TailToBegin_Fwd { ExternalAccessible := 'False'; ExternalVisible := 'False'; ExternalWritable := 'False'} : DInt;   //           Count tail to next conveyor distance
      sdi_HeadToEnd_Fwd { ExternalAccessible := 'False'; ExternalVisible := 'False'; ExternalWritable := 'False'} : DInt;   //           Count head to end distance
      sdi_TailToBegin_Rvs { ExternalAccessible := 'False'; ExternalVisible := 'False'; ExternalWritable := 'False'} : DInt;   //           Count tail to next conveyor distance
      sdi_HeadToEnd_Rvs { ExternalAccessible := 'False'; ExternalVisible := 'False'; ExternalWritable := 'False'} : DInt;   //           Count head to end distance
   END_VAR
   VAR
      sdi_PEC_EoSDistance_Fwd { ExternalAccessible := 'False'; ExternalVisible := 'False'; ExternalWritable := 'False'} : DInt;   //           Real distance between PEC and the end of distance
      sdi_PECtoEndDistance_Fwd { ExternalAccessible := 'False'; ExternalVisible := 'False'; ExternalWritable := 'False'} : DInt;   //           Distance between photeye and the end of the conveyor in cm
      sdi_PEC_EoSDistance_Rvs { ExternalAccessible := 'False'; ExternalVisible := 'False'; ExternalWritable := 'False'} : DInt;   //           Real distance between PEC and the end of distance
      sdi_PECtoEndDistance_Rvs { ExternalAccessible := 'False'; ExternalVisible := 'False'; ExternalWritable := 'False'} : DInt;   //           Distance between photeye and the end of the conveyor in cm
   END_VAR
   VAR RETAIN
      sdi_AuxEnergySave_Fwd { ExternalAccessible := 'False'; ExternalVisible := 'False'; ExternalWritable := 'False'} : DInt;   //           Auxiliary variable to calculate energy save displacement
      sdi_AuxEnergySave_Rvs { ExternalAccessible := 'False'; ExternalVisible := 'False'; ExternalWritable := 'False'} : DInt;   //           Auxiliary variable to calculate energy save displacement
      sdi_DownstreamGapTailtoHead_Fwd { ExternalAccessible := 'False'; ExternalVisible := 'False'; ExternalWritable := 'False'} : DInt;   //           Gap between the beginning of the conveyor and the closer parcel in that conveyor
      sdi_DownstreamGapHeadToHead_Fwd { ExternalAccessible := 'False'; ExternalVisible := 'False'; ExternalWritable := 'False'} : DInt;   //           Head to head between the beginning of the conveyor and the closer parcel in that conveyor
      sdi_DownstreamGapTailtoHead_Rvs { ExternalAccessible := 'False'; ExternalVisible := 'False'; ExternalWritable := 'False'} : DInt;   //           Gap between the beginning of the conveyor and the closer parcel in that conveyor
      sdi_DownstreamGapHeadToHead_Rvs { ExternalAccessible := 'False'; ExternalVisible := 'False'; ExternalWritable := 'False'} : DInt;   //           Head to head between the beginning of the conveyor and the closer parcel in that conveyor
      sdi_TransitionZone { ExternalAccessible := 'False'; ExternalVisible := 'False'; ExternalWritable := 'False'} : DInt;   // Counter of product in transition zone
   END_VAR
   VAR
      R_TRIG_ManualMode {InstructionName := 'R_TRIG'; LibVersion := '1.0'; ExternalAccessible := 'False'; ExternalVisible := 'False'; ExternalWritable := 'False'; S7_SetPoint := 'False'} : R_TRIG;   //           Rising edge trigger manual mode
      R_TRIG_Jog {InstructionName := 'R_TRIG'; LibVersion := '1.0'; ExternalAccessible := 'False'; ExternalVisible := 'False'; ExternalWritable := 'False'; S7_SetPoint := 'False'} : R_TRIG;   //           Rising edge trigger manual jog
      R_TRIG_PE_EoSFiltered_Rvs {InstructionName := 'R_TRIG'; LibVersion := '1.0'; ExternalAccessible := 'False'; ExternalVisible := 'False'; ExternalWritable := 'False'; S7_SetPoint := 'False'} : R_TRIG;   //           Rising edge trigger end of section photo eye filtered
      R_TRIG_PE_EoSFiltered_Fwd {InstructionName := 'R_TRIG'; LibVersion := '1.0'; ExternalAccessible := 'False'; ExternalVisible := 'False'; ExternalWritable := 'False'; S7_SetPoint := 'False'} : R_TRIG;   //           Rising edge trigger end of section photo eye filtered
      R_TRIG_TailToBegin_Rvs {InstructionName := 'R_TRIG'; LibVersion := '1.0'; ExternalAccessible := 'False'; ExternalVisible := 'False'; ExternalWritable := 'False'; S7_SetPoint := 'False'} : R_TRIG;   //           Rising edge trigger Tail arrive at the beginning of next conveyor
      R_TRIG_TailToBegin_Fwd {InstructionName := 'R_TRIG'; LibVersion := '1.0'; ExternalAccessible := 'False'; ExternalVisible := 'False'; ExternalWritable := 'False'; S7_SetPoint := 'False'} : R_TRIG;   //           Rising edge trigger Tail arrive at the beginning of next conveyor
      F_TRIG_ManualMode {InstructionName := 'F_TRIG'; LibVersion := '1.0'; ExternalAccessible := 'False'; ExternalVisible := 'False'; ExternalWritable := 'False'; S7_SetPoint := 'False'} : F_TRIG;   //           Falling edge trigger manual mode
      F_TRIG_Jog {InstructionName := 'F_TRIG'; LibVersion := '1.0'; ExternalAccessible := 'False'; ExternalVisible := 'False'; ExternalWritable := 'False'; S7_SetPoint := 'False'} : F_TRIG;   //           Falling edge trigger manual mode jog
      F_TRIG_PEC_EoSFiltered_Rvs {InstructionName := 'F_TRIG'; LibVersion := '1.0'; ExternalAccessible := 'False'; ExternalVisible := 'False'; ExternalWritable := 'False'; S7_SetPoint := 'False'} : F_TRIG;   //           Falling edge trigger end of section photo eye filtered
      F_TRIG_PEC_EoSFiltered_Fwd {InstructionName := 'F_TRIG'; LibVersion := '1.0'; ExternalAccessible := 'False'; ExternalVisible := 'False'; ExternalWritable := 'False'; S7_SetPoint := 'False'} : F_TRIG;   //           Falling edge trigger end of section photo eye filtered
      F_TRIG_AuxHeadToEnd_Rvs {InstructionName := 'F_TRIG'; LibVersion := '1.0'; ExternalAccessible := 'False'; ExternalVisible := 'False'; ExternalWritable := 'False'; S7_SetPoint := 'False'} : F_TRIG;   //           Falling edge trigger Aux head to end bit
      F_TRIG_AuxHeadToEnd_Fwd {InstructionName := 'F_TRIG'; LibVersion := '1.0'; ExternalAccessible := 'False'; ExternalVisible := 'False'; ExternalWritable := 'False'; S7_SetPoint := 'False'} : F_TRIG;   //           Falling edge trigger Aux head to end bit
      R_TRIG_ConveyorUp {InstructionName := 'R_TRIG'; LibVersion := '1.0'; ExternalAccessible := 'False'; ExternalVisible := 'False'; ExternalWritable := 'False'; S7_SetPoint := 'False'} : R_TRIG;   //           Rising edge trigger conveyor up time
      R_TRIG_EnergySave {InstructionName := 'R_TRIG'; LibVersion := '1.0'; ExternalAccessible := 'False'; ExternalVisible := 'False'; ExternalWritable := 'False'; S7_SetPoint := 'False'} : R_TRIG;   //           Rising edge trigger energy save
      R_TRIG_VFDRunning {InstructionName := 'R_TRIG'; LibVersion := '1.0'; ExternalAccessible := 'False'; ExternalVisible := 'False'; ExternalWritable := 'False'; S7_SetPoint := 'False'} : R_TRIG;   //           Rising edge trigger VFD running
      R_TRIG_ConveyorDownTime {InstructionName := 'R_TRIG'; LibVersion := '1.0'; ExternalAccessible := 'False'; ExternalVisible := 'False'; ExternalWritable := 'False'; S7_SetPoint := 'False'} : R_TRIG;   //           Rising edge trigger conveyor down
      R_TRIG_RunManual {InstructionName := 'R_TRIG'; LibVersion := '1.0'; ExternalAccessible := 'False'; ExternalVisible := 'False'; ExternalWritable := 'False'; S7_SetPoint := 'False'} : R_TRIG;   //           Rising edge run conveyor in manual mode
      R_TRIG_Transfering_Rvs {InstructionName := 'R_TRIG'; LibVersion := '1.0'; ExternalAccessible := 'False'; ExternalVisible := 'False'; ExternalWritable := 'False'; S7_SetPoint := 'False'} : R_TRIG;   //           Rising edge transfering
      R_TRIG_Transfering_Fwd {InstructionName := 'R_TRIG'; LibVersion := '1.0'; ExternalAccessible := 'False'; ExternalVisible := 'False'; ExternalWritable := 'False'; S7_SetPoint := 'False'} : R_TRIG;   //           Rising edge transfering
      F_TRIG_HeadAtEnd_Rvs {InstructionName := 'F_TRIG'; LibVersion := '1.0'; ExternalAccessible := 'False'; ExternalVisible := 'False'; ExternalWritable := 'False'; S7_SetPoint := 'False'} : F_TRIG;   //           Falling edge head at the end of the conveyor
      F_TRIG_HeadAtEnd_Fwd {InstructionName := 'F_TRIG'; LibVersion := '1.0'; ExternalAccessible := 'False'; ExternalVisible := 'False'; ExternalWritable := 'False'; S7_SetPoint := 'False'} : F_TRIG;   //           Falling edge head at the end of the conveyor
      R_TRIG_Reverse {InstructionName := 'R_TRIG'; LibVersion := '1.0'; ExternalAccessible := 'False'; ExternalVisible := 'False'; ExternalWritable := 'False'; S7_SetPoint := 'False'} : R_TRIG;   //           Rising edge of reverse direction
      F_TRIG_Reverse {InstructionName := 'F_TRIG'; LibVersion := '1.0'; ExternalAccessible := 'False'; ExternalVisible := 'False'; ExternalWritable := 'False'; S7_SetPoint := 'False'} : F_TRIG;   //           Falling edge of reverse direction
      R_Trig_DirectionChange {InstructionName := 'R_TRIG'; LibVersion := '1.0'; ExternalAccessible := 'False'; ExternalVisible := 'False'; ExternalWritable := 'False'; S7_SetPoint := 'False'} : R_TRIG;   //           Rising edge of change direction
      F_Trig_DirectionChange {InstructionName := 'F_TRIG'; LibVersion := '1.0'; ExternalAccessible := 'False'; ExternalVisible := 'False'; ExternalWritable := 'False'; S7_SetPoint := 'False'} : F_TRIG;   //           Falling edge of change direction
      R_TRIG_PrestartManual {InstructionName := 'R_TRIG'; LibVersion := '1.0'; ExternalAccessible := 'False'; ExternalVisible := 'False'; ExternalWritable := 'False'; S7_SetPoint := 'False'} : R_TRIG;   //   Rising edge of manual prestart
      R_TRIG_ConveyorStopped {InstructionName := 'R_TRIG'; LibVersion := '1.0'; ExternalAccessible := 'False'; ExternalVisible := 'False'; ExternalWritable := 'False'; S7_SetPoint := 'False'} : R_TRIG;   //  Rising edge of stop
      sx_Ready { ExternalAccessible := 'False'; ExternalVisible := 'False'; ExternalWritable := 'False'} : Bool;   //           Conveyor Ready to operate in Automatic mode
   END_VAR
   VAR RETAIN
      sx_StartReceived { ExternalAccessible := 'False'; ExternalVisible := 'False'; ExternalWritable := 'False'} : Bool;   //           Save start trigger from the system
      sx_EnergySaveActive { ExternalAccessible := 'False'; ExternalVisible := 'False'; ExternalWritable := 'False'} : Bool;   //           Active energy save mode
      sx_AuxHeadToEnd_Fwd { ExternalAccessible := 'False'; ExternalVisible := 'False'; ExternalWritable := 'False'} : Bool;   //           Aux bit to control head to end positioning in forward direction
      sx_AuxHeadToEnd_Rvs { ExternalAccessible := 'False'; ExternalVisible := 'False'; ExternalWritable := 'False'} : Bool;   //           Aux bit to control head to end positioning in reverse direction
      sx_TailToBegin_Fwd { ExternalAccessible := 'False'; ExternalVisible := 'False'; ExternalWritable := 'False'} : Bool;   //           Tail to begin done in forward direction
      sx_TailToBegin_Rvs { ExternalAccessible := 'False'; ExternalVisible := 'False'; ExternalWritable := 'False'} : Bool;   //           Tail to begin done in reverse direction
      sx_Gapping_Fwd { ExternalAccessible := 'False'; ExternalVisible := 'False'; ExternalWritable := 'False'} : Bool;   //           Gapping in process in forward direction
      sx_Gapping_Rvs { ExternalAccessible := 'False'; ExternalVisible := 'False'; ExternalWritable := 'False'} : Bool;   //           Gapping in process in reverse direction
   END_VAR
   VAR
      sx_AutomaticActive { ExternalAccessible := 'False'; ExternalVisible := 'False'; ExternalWritable := 'False'} : Bool;   //           Automatic active
   END_VAR
   VAR RETAIN
      sx_RecoveryGap_Fwd { ExternalAccessible := 'False'; ExternalVisible := 'False'; ExternalWritable := 'False'} : Bool;   //           Recovery gap activated in forward direction
      sx_RecoveryGap_Rvs { ExternalAccessible := 'False'; ExternalVisible := 'False'; ExternalWritable := 'False'} : Bool;   //           Recovery gap activated in reverse direction
   END_VAR
   VAR
      sx_ManualModeActive { ExternalAccessible := 'False'; ExternalVisible := 'False'; ExternalWritable := 'False'} : Bool;   //           Manual mode active
      sx_PreStartManual { ExternalAccessible := 'False'; ExternalVisible := 'False'; ExternalWritable := 'False'} : Bool;   //           Pre conditions to run conveyor in manual mode
   END_VAR
   VAR RETAIN
      sx_AuxHeadAtEnd_Fwd { ExternalAccessible := 'False'; ExternalVisible := 'False'; ExternalWritable := 'False'} : Bool;   //           Parcel reach the end of the conveyor in forward direction
      sx_AuxHeadAtEnd_Rvs { ExternalAccessible := 'False'; ExternalVisible := 'False'; ExternalWritable := 'False'} : Bool;   //           Parcel reach the end of the conveyor in reverse direction
   END_VAR
   VAR
      sx_CascadeStartUp { ExternalAccessible := 'False'; ExternalVisible := 'False'; ExternalWritable := 'False'} : Bool;   //           Cascade startup auxiliary bit
      sx_DirectionChanged { ExternalAccessible := 'False'; ExternalVisible := 'False'; ExternalWritable := 'False'} : Bool;   //           Change direction until stop
      sx_ReverseDirection { ExternalAccessible := 'False'; ExternalVisible := 'False'; ExternalWritable := 'False'} : Bool;   //           Direction Selection auxiliary bit
      sx_ManualRunning { ExternalAccessible := 'False'; ExternalVisible := 'False'; ExternalWritable := 'False'} : Bool;   //          Conveyor running in manual mode
      sx_Up { ExternalAccessible := 'False'; ExternalVisible := 'False'; ExternalWritable := 'False'} : Bool;   //  Conveyor is up
      sx_Down { ExternalAccessible := 'False'; ExternalVisible := 'False'; ExternalWritable := 'False'} : Bool;   //  Conveyor is down
      sx_Stopped { ExternalAccessible := 'False'; ExternalVisible := 'False'; ExternalWritable := 'False'} : Bool;   //  Conveyor is stopped
      si_EnergySaveFilter { ExternalAccessible := 'False'; ExternalVisible := 'False'; ExternalWritable := 'False'} : Int;   // Energy save filter distance
   END_VAR

   VAR_TEMP
      tx_CascadeStart : Bool;
   END_VAR

   VAR CONSTANT
      ci_OverflowLimit : Int := 32000;   //           Limit int overflow
      ci_MinimumParcelLength : Int := 13;   // Minimum parcel length [cm]
   END_VAR


BEGIN

	(*
	----------------------------------------------------------------------------------------
	|                                                                                      |
	|  Copyright  2019             MHS Europe BV                                           |
	|  All Rights Rese9ved         Larenweg 90                                             |
	|                              5234 KC 's-Hertogenbosch,                               |
	|                              Netherlands                                             |
	|                                                                                      |
	----------------------------------------------------------------------------------------

	Version history:
	Date        | Version   | Author        | Remark
	----------------------------------------------------------------------------------------
	            | 3.0       | C.Leite       | First release TIA 15.1
	01/01/2020  | 3.1       | S. Deulkar    | Modified error loging, added reset to reset internal error
	                                        | Cosidered commissioning error to put conveyor in ready state
	07/01/2020  | 3.2       | C. Leite      | Manual mode bug corrected related with conveyor start
	10/01/2020  | 3.3       | C. Leite      | Manual mode start\stop change
	                                        | Lenght conveyor data type was changed to DInt
	14/01/2020  | 3.4       | F.Baten       | Renamed Trail to Tail
	                                        | Renamed ii_PEC_EosDistance_EoS to idi_PEC_EoSDistance same for BoS
	21/01/2020  | 3.5       | C.Leite       | Reset gapping bits when the direction changes
	06/01/2020  | 3.6       | S. Deulkar    | Added safety Ok in condition to make ready status
	25/02/2020  | 3.7       | S. Deulkar    | Modified to update ststus output every cycle
	21/04/2020  | 3.8       | F.Baten       | Modified energysave reset
	23/04/2020  | 3.9       | S. Deulkar    | Modified logic for reset energy save command if it is slave conveyor
	22/06/2020  | 3.10      | K. Pokorski   | Modified singaling request activation, modified stop conditions (Handshake ReqStop)
	02/07/2020  | 3.11      | K. Pokorski   | Modified condition to disable manual mode (safety ok)
	30/07/2020  | 3.12      | S. Theocharis | Reset HMI commands of manual mode when conveyor no ready
	                                        | Keep downstream running when the a PEC error occurs
	04/08/2020  | 3.13      | S. Deulkar    | Deletded Manual run stop command and Modified code to let
	                                        | let slave conveyor go in energy save, Optimized energy save logic
	17/08/2020  | 3.14      | L.Klar        | Gapping corrected to work with PEC offset. Gap correction configuration added
	17/08/2020  | 3.15      | S. Theocharis | Encoder fault added. Manual mode active to interface. Stop trigger added for statistics
	                                        | Fix  statistics
	11/01/2021  | 3.16      | L.Klar        | Input safety ok added to stop conveyor condition
	02/03/2021  | 3.17      | K. Pokorski   | Halted status enable only when automatic on
	11/03/2021  | 3.18      | S. Theocharis | Added bulk flow mode 3
	13/03/2021  | 3.19      | S. Theocharis | Warning color commented, line 665 added, sensors initial values changed to true
	15/03/2021  | 3.20      | S. Theocharis | Energy safe corrected
	29/03/2021  | 3.21      | M. Kocot      | Added HMI command for manual speed percetage selection and modified logic for cascade
	                                        | startup
	31/03/2021  | 3.22      | H.Rutkowski   | Changed logic for TransitionZone calculation in mode 3( Converted PEC distance to cm)
	14/05/2021  | 3.23      | S. Nikodem    | Reset value from iq_UDT_HandShakeUp.DownstreamDisplacement and iq_UDT_HandShake.DownstreamDisplacement
	28/06/2021  | 3.24      | N.Kadam       | Modified logic for conveyor downtime and Esave statistics
	29/07/2021  | 3.25      | S. Deulkar    | Autotic ON condition is added to excecut region 7: Automatic mode active
	                                        | Statistics are updated after status
	11/11/2021  | 3.26      | M.Singh       |Shared Hardware signal over Interface
	28/03/2022  | 3.27      | M.Singh       |Solved Esave Bug, Swapped regions "Operation modes" and "Energy Save"
	28/07/2022  | 3.28      | M.Singh       |Removed handsakeUP.RTR from conditions determining downstream TIP and RTS
	30/07/2022  | 3.28      | M.Singh       |Addded hardware ok as condition to show safety status
	                                        |Added Aux Head at end and TIP to Esave Reset conditions
	11.08.2023  | 3.29      | M.Diebel      |Comment logic to set #s_UDT_CommonStatus.Warning
	08.09.2023  | 3.30      | M.Diebel      |Updated Lenght for transition Zone in reverse direction
	05.10.2023  | 3.31      | M.Diebel      |Updated Reset Energe Save in reverse direction
	20.12.2023  | 3.32      | M.Diebel      |Reset Energy save in reverse direction
	31.01.2024  | 3.33      | L.Klar        |Energy save filter added
	*)

	REGION 1 - Initial

	    REGION 1.1 - First PLC cycle

	        // Conveyor stops in the first scan of the PLC
	        IF "DB_Memory".FirstScan
	        THEN
	            #iq_UDT_EquipmentControl.Command.Start := FALSE;    // Command start
	            #sx_AutomaticActive := FALSE;                       // switch of automatic active
	            #iq_UDT_HandShakeUp.RTR := False;                   // Reset RTR signal

	            #iq_UDT_HandShakeUp.CascadeStartUp := FALSE;        // Reset cascade start signal

	            #iq_UDT_ConveyorInterface.RunFwd := FALSE;          // Order to run forward to VFD
	            #iq_UDT_ConveyorInterface.RunRvs := FALSE;          // Order to run reverse to VFD

	        END_IF;

	    END_REGION

	    REGION 1.2 - Conversion distance between PEC and end of conveyor [mm to cm]

	        // Move PEC Distance into a static variable. Added on version 2.8
	        #sdi_PEC_EoSDistance_Fwd := #idi_PEC_EoSDistance;
	        #sdi_PEC_EoSDistance_Rvs := #i_UDT_ConveyorConfiguration.Common.Length - #idi_PEC_BoSDistance;

	        // Limit to prevent malfunctions with zero or negative values. Added on version 2.8
	        IF #sdi_PEC_EoSDistance_Fwd < 10
	        THEN
	            #sdi_PEC_EoSDistance_Fwd := 10;
	        END_IF;

	        IF #sdi_PEC_EoSDistance_Rvs < 10
	        THEN
	            #sdi_PEC_EoSDistance_Rvs := 10;
	        END_IF;

	        //  Convertion of the distance between photo eye and the end of the conveyor from mm to cm.
	        #sdi_PECtoEndDistance_Fwd := (#sdi_PEC_EoSDistance_Fwd
	        - #i_UDT_ConveyorConfiguration.Forward_Direction.PEC_EoSDistanceOffset) / 10;

	        #sdi_PECtoEndDistance_Rvs := (#sdi_PEC_EoSDistance_Rvs
	        - #i_UDT_ConveyorConfiguration.Reverse_Direction.PEC_BoSDistanceOffset) / 10;


	        // Limit the Pec to End distance in positive ranges. Added on version 2.7
	        IF #sdi_PECtoEndDistance_Fwd < 1 THEN
	            #sdi_PECtoEndDistance_Fwd := 1;
	        END_IF;

	        IF #sdi_PECtoEndDistance_Rvs < 1 THEN
	            #sdi_PECtoEndDistance_Rvs := 1;
	        END_IF;

	        #sx_ReverseDirection := (#iq_UDT_ConveyorCommand.Reverse OR #ix_ReverseDirection) AND #i_UDT_ConveyorConfiguration.Bi_Directional_Enable;


	    END_REGION

	    REGION 1.3 Conditions Up - Down - Stopped
	        //Used for statistics

	        #sx_Up := (#sx_AutomaticActive                               // Automatic active
	        AND #sx_Ready                                                // Ready active
	        AND NOT #sx_EnergySaveActive);                              // Not in energy save

	        #sx_Down := (NOT #sx_ManualModeActive                                                   // Not in manual mode
	        AND #s_UDT_CommonStatus.Error                                                           // in error
	        AND NOT #sx_Ready                                                                       // Conveyor not ready
	        AND NOT #sx_EnergySaveActive);                                                          // Not in energy save

	        #sx_Stopped := (NOT #sx_AutomaticActive AND #sx_Ready);

	    END_REGION

	    REGION 1.3 - Triggers

	        // Rising edge trigger manual mode
	        #R_TRIG_ManualMode(CLK := #iq_UDT_ConveyorCommand.ManualMode
	                           OR #iq_UDT_EquipmentControl.Command.ManualMode);

	        // Falling edge trigger manual mode
	        #F_TRIG_ManualMode(CLK := #iq_UDT_ConveyorCommand.ManualMode
	                           OR #iq_UDT_EquipmentControl.Command.ManualMode);

	        // Rising edge trigger manual mode jog
	        #R_TRIG_Jog(CLK := #iq_UDT_ConveyorCommand.ManualJog);

	        // Falling edge trigger manual mode jog
	        #F_TRIG_Jog(CLK := #iq_UDT_ConveyorCommand.ManualJog);

	        // Rising edge trigger to start in manual mode
	        #R_TRIG_RunManual(CLK := #iq_UDT_ConveyorCommand.ManualStartStop);

	        // Rising edge trigger end of section photo eye filtered
	        #R_TRIG_PE_EoSFiltered_Fwd(CLK := #ix_PEC_EoS);
	        #R_TRIG_PE_EoSFiltered_Rvs(CLK := #ix_PEC_BoS);

	        // Falling edge trigger end of section photo eye filtered
	        #F_TRIG_PEC_EoSFiltered_Fwd(CLK := #ix_PEC_EoS);
	        #F_TRIG_PEC_EoSFiltered_Rvs(CLK := #ix_PEC_BoS);

	        // Rising edge conveyor up
	        #R_TRIG_ConveyorUp(CLK := #sx_Up);

	        // Rising edge energy save mode
	        #R_TRIG_EnergySave(CLK := #sx_EnergySaveActive);

	        // Rising edge running
	        #R_TRIG_VFDRunning(CLK := #iq_UDT_ConveyorInterface.VFDRunning);

	        // Rising edge conveyor conveyor down
	        #R_TRIG_ConveyorDownTime(CLK := #sx_Down);

	        //Rising edge conveyor stopped
	        #R_TRIG_ConveyorStopped(CLK := #sx_Stopped);

	        // Rising edge conveyor command reverse direction
	        #R_TRIG_Reverse(CLK := #iq_UDT_ConveyorCommand.Reverse);

	        // Falling edge conveyor command reverse direction
	        #F_TRIG_Reverse(CLK := #iq_UDT_ConveyorCommand.Reverse);

	        // Rising edge conveyor change direction
	        #R_Trig_DirectionChange(CLK := #sx_ReverseDirection);

	        // Falling edge conveyor change direction
	        #F_Trig_DirectionChange(CLK := #sx_ReverseDirection);

	    END_REGION

	    REGION 1.4 - Move displacement to upstream

	        // Downstream displacement is mode to upstream conveyor to calculate gap

	        IF NOT #sx_ReverseDirection
	        THEN
	            #iq_UDT_HandShakeUp.DownstreamDisplacement := #iq_UDT_ConveyorInterface.Displacement;
	        ELSE
	            #iq_UDT_HandShake.DownstreamDisplacement := #iq_UDT_ConveyorInterface.Displacement;

	        END_IF;

	    END_REGION

	    REGION 1.5 - Change direction

	        // The memory bit to change direction is activated when the input is trigger

	        IF #R_Trig_DirectionChange.Q
	            OR #F_Trig_DirectionChange.Q
	        THEN
	            #sx_DirectionChanged := TRUE;
	        END_IF;

	        // The direction changed memory bit is just reset when the conveyor stops to prevente mechanical problems

	        IF #sx_DirectionChanged
	            AND #i_UDT_ConveyorConfiguration.Bi_Directional_Enable
	            AND NOT #iq_UDT_ConveyorInterface.VFDatSpeed
	            AND NOT #iq_UDT_ConveyorInterface.VFDRunning
	            AND (#iq_UDT_ConveyorInterface.ActualSpeed <= 0)
	        THEN
	            #sx_DirectionChanged := FALSE;

	            #sx_AuxHeadAtEnd_Fwd := FALSE;
	            #sx_AuxHeadAtEnd_Rvs := FALSE;

	            #sdi_AuxGapHeadToHeadCounter_Fwd := 0;
	            #sdi_AuxGapHeadToHeadCounter_Rvs := 0;

	            #sdi_AuxGapTailtoHeadCounter_Rvs := 0;
	            #sdi_AuxGapTailtoHeadCounter_Fwd := 0;

	            #sx_Gapping_Rvs := FALSE;
	            #sx_Gapping_Fwd := FALSE;

	            #iq_UDT_HandShake.TIP := FALSE;
	            #iq_UDT_HandShakeUp.TIP := FALSE;

	            #iq_UDT_HandShakeUp.DownstreamDisplacement := 0;     // v3.23
	            #iq_UDT_HandShake.DownstreamDisplacement := 0;       // v3.23

	        END_IF;

	        IF (#R_Trig_DirectionChange.Q
	            AND NOT #ix_PEC_BoS)
	            OR (#F_Trig_DirectionChange.Q
	            AND NOT #ix_PEC_EoS)
	            AND #i_UDT_ConveyorConfiguration.Bi_Directional_Enable
	        THEN
	            #sdi_AuxGapHeadToHeadCounter_Fwd := 0;
	            #sdi_AuxGapHeadToHeadCounter_Rvs := 0;
	        END_IF;

	    END_REGION

	    REGION 1.5 - Gaps configuration

	        // Forward head to head
	        #sdi_GapHeadToHeadConfiguration_Fwd := #i_UDT_ConveyorConfiguration.Forward_Direction.GapHeadToHead + #i_UDT_ConveyorConfiguration.Forward_Direction.GapCorrection;
	        // Forward tail to head
	        #sdi_GapTailToHeadConfiguration_Fwd := #i_UDT_ConveyorConfiguration.Forward_Direction.GapTailToHead + #i_UDT_ConveyorConfiguration.Forward_Direction.GapCorrection;
	        // Reverse head to head
	        #sdi_GapHeadToHeadConfiguration_Rvs := #i_UDT_ConveyorConfiguration.Reverse_Direction.GapHeadToHead + #i_UDT_ConveyorConfiguration.Reverse_Direction.GapCorrection;
	        // Reverse tail to head
	        #sdi_GapTailToHeadConfiguration_Rvs := #i_UDT_ConveyorConfiguration.Reverse_Direction.GapTailToHead + #i_UDT_ConveyorConfiguration.Reverse_Direction.GapCorrection;

	    END_REGION

	END_REGION

	REGION 2 - Reset faults

	    REGION 2.1 - Send reset request to interface UDT

	        // Reset signal is sent to the interface UDT (VFD block, Tracking block, PEC update block)
	        #iq_UDT_ConveyorInterface.InternalErrorReset := #iq_UDT_EquipmentControl.Command.Reset;

	        #iq_UDT_ConveyorInterface.ResetStatistics := #iq_UDT_EquipmentControl.Command.ResetData;

	    END_REGION


	    REGION 2.2 - Error / warning

	        #s_UDT_CommonStatus.Error := #iq_UDT_ConveyorInterface.InternalErrorPEC               // Internal PEC error status
	        OR #iq_UDT_ConveyorInterface.InternalErrorVFD               // Internal VFD error status
	        OR #iq_UDT_ConveyorInterface.InternalErrorTracking          // Internal tracking error status
	        OR #iq_UDT_ConveyorInterface.Disconnected                   // Isolator switch error status
	        OR #iq_UDT_ConveyorInterface.InternalErrorEncoder;          // Encoder error


	        // #s_UDT_CommonStatus.Warning := #iq_UDT_ConveyorInterface.InternalWarningTracking        // v2.3 Internal Warning Tracking  added
	        // OR #iq_UDT_ConveyorInterface.InternalWarningVFD;                                        // v2.3 Internal Warning VFD added

	    END_REGION

	END_REGION

	REGION 3 - Check conditions to set conveyor ready
	    //Share HardwareOK signal over interface
	    #iq_UDT_ConveyorInterface.HardwareOk := #ix_HardwareOk;

	    //  Conditions to set bit sx_Ready to operate in automatic mode
	    #sx_Ready := NOT #s_UDT_CommonStatus.Error                              // Ready bit is set true when common error status its false
	    AND #ix_SafetyOk
	    AND #ix_24vOk                                                        // 24V error status
	    AND #ix_400vOk                                                       // 400V error status
	    AND #ix_HardwareOk                                                   // Profinet error status
	    AND NOT #iq_UDT_ConveyorInterface.ConfigurationError;                // No configuration error

	END_REGION

	REGION 4 - Stop conveyor

	    // Conditions to stop conveyor
	    IF (#F_TRIG_Jog.Q                                           // Trigger when conveyor stops jogging by HMI
	        AND #sx_ManualModeActive)                                   // Manual mode is active

	        OR (NOT #iq_UDT_EquipmentControl.Command.AutomaticOn        // Conveyor stops if the bit AutomaticOn from control block is false
	        AND NOT #sx_ManualModeActive)                               // Manual mode active bit

	        OR (NOT #sx_Ready                                           // Bit conveyor ready to run in automatic mode
	        AND NOT #sx_ManualModeActive)                               // Manual mode active

	        OR #R_TRIG_ManualMode.Q                                     // Trigger when manual mode is set on
	        OR #F_TRIG_ManualMode.Q                                     // Trigger when manual mode is set off

	        OR (#iq_UDT_HandShakeUp.ReqStop                             // Stop request from upstream if direction not changed
	        AND NOT #sx_DirectionChanged)

	        OR (#iq_UDT_HandShake.ReqStop                               // Stop request from downstream if direction changed
	        AND #sx_DirectionChanged)

	        OR NOT #ix_SafetyOk

	    THEN
	        //  Order to stop VFD
	        #iq_UDT_ConveyorInterface.RunFwd := FALSE;                  // Set false order to VFD run in forward direction
	        #iq_UDT_ConveyorInterface.RunRvs := FALSE;                  // Set false order to VFD run in reverse direction

	        IF NOT #sx_ReverseDirection
	        THEN

	            #iq_UDT_HandShakeUp.RTR := FALSE;                       // Set false the bit ready to receive
	            #iq_UDT_HandShakeUp.CascadeStartUp := FALSE;            // Set false cascade start up bit

	        ELSE

	            #iq_UDT_HandShake.RTR := FALSE;                       // Set false the bit ready to receive
	            #iq_UDT_HandShake.CascadeStartUp := FALSE;            // Set false cascade start up bit

	        END_IF;

	        #sx_AutomaticActive := FALSE;                               // Automatic mode is disable
	        //    #sx_StartReceived := FALSE;                                 // Clear start receive bit

	    END_IF;

	END_REGION

	REGION 5 - Start

	    REGION 5.1 - Save Start bit request

	        // The conditions to set the bit "startReceived" are:
	        // - Conveyor not in manual mode.
	        // - Conveyor ready to run.
	        // - Bit AutomaticOn from control block must be on.
	        // - Bit start form control block on.

	        IF #iq_UDT_EquipmentControl.Command.Start
	            AND #iq_UDT_EquipmentControl.Command.AutomaticOn
	        THEN
	            #sx_StartReceived := TRUE;          // Start bit from control block received
	        END_IF;

	    END_REGION

	    REGION 5.2 - Cascade mode

	        (* If the bit "StartReceived" is set, automatic mode is activated if the conveyor is set as the first one to run
	         or the bit cascadestartup from downstream is on. *)

	        IF #iq_UDT_EquipmentControl.Command.Start
	            AND #iq_UDT_EquipmentControl.Command.AutomaticOn
	            AND NOT #sx_ManualModeActive
	            AND #sx_Ready
	        THEN
	            #sx_AutomaticActive := TRUE;        // Conveyor active automatic mode
	        END_IF;

	        //Timer to cascade mode
	        #tx_CascadeStart := #sx_StartReceived
	        AND ((NOT #sx_ReverseDirection
	        AND (#i_UDT_ConveyorConfiguration.Forward_Direction.FirstConveyorToStart
	        OR #iq_UDT_HandShake.CascadeStartUp))
	        OR (#sx_ReverseDirection
	        AND (#i_UDT_ConveyorConfiguration.Reverse_Direction.FirstConveyorToStart
	        OR #iq_UDT_HandShakeUp.CascadeStartUp)));

	        #s_FB_CascadeModeTimer(iudi_OnDelayTime := #i_UDT_ConveyorConfiguration.CascadeTimeOnDelay,      // Cascade mode timer
	                               ix_SignalToDelay := #tx_CascadeStart,
	                               ix_Enable := TRUE,                                                   // Signal ready to enable cascade mode
	                               qx_DelayedSignal => #sx_CascadeStartUp);

	        IF NOT #iq_UDT_EquipmentControl.Command.AutomaticOn
	        THEN
	            #sx_StartReceived := False;
	        END_IF;


	        // Cascade mode signal to upstream
	        IF NOT #sx_ReverseDirection
	        THEN
	            #iq_UDT_HandShakeUp.CascadeStartUp := #sx_CascadeStartUp;
	        ELSE
	            #iq_UDT_HandShake.CascadeStartUp := #sx_CascadeStartUp;
	        END_IF;



	    END_REGION

	END_REGION

	REGION 6 - Manual mode

	    REGION 6.1 - Manual mode force disable

	        // Manual mode bits inputs can be reset in case of malfunction
	        IF #iq_UDT_EquipmentControl.Command.DisableManualMode
	        THEN
	            #iq_UDT_ConveyorCommand.ManualMode := False;
	            #iq_UDT_EquipmentControl.Command.ManualMode := False;
	        END_IF;

	    END_REGION

	    REGION 6.2 - Manual mode activation

	        // Manual mode is active if it is active from hmi or by control block
	        #sx_ManualModeActive := #iq_UDT_ConveyorCommand.ManualMode
	        OR #iq_UDT_EquipmentControl.Command.ManualMode;

	        //Send manual mode active to PEC/VFD blocks to supress errors
	        #iq_UDT_ConveyorInterface.ManualModeActive := #sx_ManualModeActive;

	    END_REGION

	    REGION 6.3 - Reset manual commands
	        //When the system is not any more in manual mode or when fatal error occurs the HMI commands should be reset
	        //Added in V3.12 as bug fix.
	        IF NOT #ix_SafetyOk
	            OR NOT #ix_24vOk                                                        // 24V error status
	            OR NOT #ix_400vOk                                                       // 400V error status
	            OR NOT #ix_HardwareOk                                                   // Profinet error status
	            OR #iq_UDT_ConveyorInterface.ConfigurationError                          // No configuration err
	            OR #iq_UDT_ConveyorInterface.InternalErrorVFD
	            OR #iq_UDT_ConveyorInterface.Disconnected
	            OR NOT #sx_ManualModeActive
	        THEN
	            #iq_UDT_ConveyorCommand.ManualStartStop := FALSE;
	            #iq_UDT_ConveyorCommand.ManualFullSpeed := FALSE;
	            #iq_UDT_ConveyorCommand.ManualJog := FALSE;
	            #iq_UDT_ConveyorCommand.Reverse := FALSE;
	        END_IF;

	    END_REGION

	    REGION 6.4 - Start/Stop

	        // Pre start conditions to run in manual mode
	        #sx_PreStartManual := #sx_ManualModeActive              // Manual mode active bit
	        AND #ix_SafetyOk                                        // Safety healthy bit
	        AND NOT #iq_UDT_ConveyorInterface.Disconnected          // Isolator switch connected
	        AND #ix_HardwareOk                                      // Profinet comunication
	        AND NOT #iq_UDT_ConveyorInterface.InternalErrorVFD;     // Internal error from VFD

	        #R_TRIG_PrestartManual(CLK := #sx_PreStartManual);


	        IF (#sx_PreStartManual                                  // Pre start conditions to run in manual mode
	            AND (#R_TRIG_RunManual.Q                            // Trigger when conveyor start running in manual mode
	            OR (#iq_UDT_ConveyorCommand.ManualStartStop             // Conveyor start running in manual mode active
	            AND #R_TRIG_PrestartManual.Q)                       // Trigger when pre start conditions ti run in manual mode
	            AND NOT #iq_UDT_ConveyorCommand.ManualJog)          // Conveyor is not running in jog
	            OR (#sx_PreStartManual AND #R_TRIG_Jog.Q                                   // Trigger to start jogging
	            AND NOT #iq_UDT_ConveyorCommand.ManualStartStop))       // Conveyor is not running in manual mode
	        THEN

	            #iq_UDT_EquipmentControl.Request.SignalingRequest := TRUE;  // Request signaling to control block before conveyor run in manual mode

	        END_IF;

	        // Run conveyor forward in manual mode
	        #iq_UDT_ConveyorInterface.RunFwd := #sx_PreStartManual           // Pre start conditions to run in manual mode
	        AND NOT #iq_UDT_ConveyorCommand.Reverse                          // Not in reverse direction
	        AND (NOT #iq_UDT_EquipmentControl.Request.SignalingRequest       // Signaling request done
	        OR #sx_ManualRunning)
	        AND (#iq_UDT_ConveyorCommand.ManualStartStop                         // Manual mode start to run
	        OR #iq_UDT_ConveyorCommand.ManualJog);                           // Jogging

	        // Run conveyor reverse in manual mode
	        #iq_UDT_ConveyorInterface.RunRvs := #sx_PreStartManual           // Pre start conditions to run in manual mode
	        AND #iq_UDT_ConveyorCommand.Reverse                              // Reverse direction
	        AND (NOT #iq_UDT_EquipmentControl.Request.SignalingRequest       // Signaling request done
	        OR #sx_ManualRunning)
	        AND (#iq_UDT_ConveyorCommand.ManualStartStop                         // Manual mode start to run
	        OR #iq_UDT_ConveyorCommand.ManualJog);                           // Jogging

	        #sx_ManualRunning := #iq_UDT_ConveyorInterface.RunFwd
	        OR #iq_UDT_ConveyorInterface.RunRvs;

	    END_REGION

	END_REGION

	REGION 7 - Automatic mode active

	    IF NOT #sx_ManualModeActive // Manual mode is not active
	    THEN
	        REGION 7.1 - Head to End

	            (*  Function to calculate when the head of the parcel reaches the end of the conveyor
	                When PEC detects parcels head, the functionality increments the displacement of the conveyor until reach the value of the distance
	                between PEC and the end of the conveyor. After that, the counter is reset and the bit #sx_AuxHeadToEnd is triggered to inform the system. *)
	            IF NOT #sx_ReverseDirection
	            THEN
	                REGION 7.1.1 - Forward

	                    IF #F_TRIG_PEC_EoSFiltered_Fwd.Q      // Detects the product's head
	                    THEN

	                        #sdi_HeadToEnd_Fwd := #sdi_PECtoEndDistance_Fwd;                // move the distance between PE and the end of the conveyor to auxiliary variable
	                        #sx_AuxHeadToEnd_Fwd := TRUE;                             // Active head to end function

	                        #sdi_GapHeadToHead_Fwd := #sdi_AuxGapHeadToHeadCounter_Fwd;     // Move gap calculated to variable
	                        #sdi_AuxGapHeadToHeadCounter_Fwd := 0;                     // Reset gap counter

	                        #sdi_Gap_Fwd := #sdi_AuxGapTailtoHeadCounter_Fwd;    // Move gap calculated to variable
	                        #sdi_AuxGapTailtoHeadCounter_Fwd := 0;                     // Reset gap counter

	                        #iq_UDT_HandShake.RTS := TRUE;                         // Set ready to send true when a parcel is detected in the PEC

	                    END_IF;

	                    IF #sx_AuxHeadToEnd_Fwd                 // Parcel's head detected in photo cell
	                        AND (#sdi_HeadToEnd_Fwd > 0)         // Psrcel's head do not arrive in the end of the conveyor yet
	                    THEN

	                        #sdi_HeadToEnd_Fwd -= #iq_UDT_ConveyorInterface.Displacement;   // Count displacement until arrive to the end of the conveyor

	                    ELSE

	                        #sx_AuxHeadToEnd_Fwd := FALSE;      // Stop function head to end

	                    END_IF;

	                    // Falling edge trigger Aux Head to End bit
	                    #F_TRIG_AuxHeadToEnd_Fwd(CLK := #sx_AuxHeadToEnd_Fwd);

	                    IF #F_TRIG_AuxHeadToEnd_Fwd.Q
	                    THEN
	                        #sx_AuxHeadAtEnd_Fwd := TRUE;                       // The head of the parcel is at the front positon of the conveyor
	                    END_IF;


	                    #F_TRIG_HeadAtEnd_Fwd(CLK := #sx_AuxHeadAtEnd_Fwd);

	                END_REGION
	            ELSE
	                REGION 7.1.2 - Reverse

	                    IF #F_TRIG_PEC_EoSFiltered_Rvs.Q      // Detects the product's head
	                    THEN

	                        #sdi_HeadToEnd_Rvs := #sdi_PECtoEndDistance_Rvs;                // move the distance between PE and the end of the conveyor to auxiliary variable
	                        #sx_AuxHeadToEnd_Rvs := TRUE;                             // Active head to end function

	                        #sdi_GapHeadToHead_Rvs := #sdi_AuxGapHeadToHeadCounter_Rvs;     // Move gap calculated to variable
	                        #sdi_AuxGapHeadToHeadCounter_Rvs := 0;                     // Reset gap counter

	                        #sdi_Gap_Rvs := #sdi_AuxGapTailtoHeadCounter_Rvs;    // Move gap calculated to variable
	                        #sdi_AuxGapTailtoHeadCounter_Rvs := 0;                     // Reset gap counter

	                        #iq_UDT_HandShakeUp.RTS := TRUE;                         // Set ready to send true when a parcel is detected in the PEC

	                    END_IF;

	                    IF #sx_AuxHeadToEnd_Rvs                 // Parcel's head detected in photo cell
	                        AND (#sdi_HeadToEnd_Rvs > 0)         // Psrcel's head do not arrive in the end of the conveyor yet
	                    THEN

	                        #sdi_HeadToEnd_Rvs += #iq_UDT_ConveyorInterface.Displacement;   // Count displacement until arrive to the end of the conveyor

	                    ELSE

	                        #sx_AuxHeadToEnd_Rvs := FALSE;      // Stop function head to end

	                    END_IF;

	                    // Falling edge trigger Aux Head to End bit
	                    #F_TRIG_AuxHeadToEnd_Rvs(CLK := #sx_AuxHeadToEnd_Rvs);

	                    IF #F_TRIG_AuxHeadToEnd_Rvs.Q
	                    THEN
	                        #sx_AuxHeadAtEnd_Rvs := TRUE;                       // The head of the parcel is at the front positon of the conveyor
	                    END_IF;


	                    #F_TRIG_HeadAtEnd_Rvs(CLK := #sx_AuxHeadAtEnd_Rvs);

	                END_REGION
	            END_IF;
	        END_REGION

	        REGION 7.2 - Tail to Begin

	            (*   This function tracks when parcels tail reaches the begin of downstream conveyor
	                 When the PEC is clear, the function start to increase the displacement until reaches the distance
	                 between PEC and the end of conveyor. *)
	            IF NOT #sx_ReverseDirection
	            THEN
	                REGION 7.2.1 - Forward

	                    IF #R_TRIG_PE_EoSFiltered_Fwd.Q                     // Detects product's tail
	                    THEN

	                        #sdi_TailToBegin_Fwd := (#sdi_PEC_EoSDistance_Fwd / 10);   // move distance between PE and the end of the conveyor to auxiliar variable

	                    END_IF;

	                    IF (#sdi_TailToBegin_Fwd > 0)                                           // While tails parcel do not reach the beginning of next conveyor
	                    THEN

	                        #sdi_TailToBegin_Fwd -= #iq_UDT_ConveyorInterface.Displacement;   // count displacement until the product's tail arrive to the next conveyor
	                        #sx_TailToBegin_Fwd := FALSE;                                    // Reset tail to begin bit

	                    ELSE

	                        #sx_TailToBegin_Fwd := TRUE;                                     // Product's tail arrived at the begin OF next conveyor

	                    END_IF;

	                    // Rising edge trigger Aux tail to Begin bit
	                    #R_TRIG_TailToBegin_Fwd(CLK := #sx_TailToBegin_Fwd);

	                END_REGION
	            ELSE
	                REGION 7.2.2 - Reverse

	                    IF #R_TRIG_PE_EoSFiltered_Rvs.Q                     // Detects product's tail
	                    THEN

	                        #sdi_TailToBegin_Rvs := (#sdi_PEC_EoSDistance_Rvs / 10);   // move distance between PE and the end of the conveyor to auxiliar variable

	                    END_IF;

	                    IF (#sdi_TailToBegin_Rvs > 0)                                           // While tails parcel do not reach the beginning of next conveyor
	                    THEN

	                        #sdi_TailToBegin_Rvs += #iq_UDT_ConveyorInterface.Displacement;   // count displacement until the product's tail arrive to the next conveyor
	                        #sx_TailToBegin_Rvs := FALSE;                                    // Reset tail to begin bit

	                    ELSE

	                        #sx_TailToBegin_Rvs := TRUE;                                     // Product's tail arrived at the begin OF next conveyor

	                    END_IF;

	                    // Rising edge trigger Aux tail to Begin bit
	                    #R_TRIG_TailToBegin_Rvs(CLK := #sx_TailToBegin_Rvs);

	                END_REGION
	            END_IF;
	        END_REGION

	        REGION 7.3 - Gap

	            (*    Gap tail TO head function calculates the distance (Gap) between two parcels.
	                  The function increases the Counter WHILE the photo eye is clear.
	                  Everytime a parcel trigger the photo eye, gap value is save AND the counter is reset.  *)
	            IF NOT #sx_ReverseDirection
	            THEN
	                REGION 7.3.1 - Forward

	                    IF #ix_PEC_EoS       // Count displacement when the PE do not detects the product
	                    THEN

	                        IF #sdi_AuxGapTailtoHeadCounter_Fwd < #ci_OverflowLimit        // Prevent integer variable overflow
	                        THEN
	                            IF #iq_UDT_HandShake.RTR THEN
	                                #sdi_AuxGapTailtoHeadCounter_Fwd += #iq_UDT_ConveyorInterface.Displacement;    // Calculate the gap
	                            END_IF;

	                        END_IF;

	                    END_IF;

	                END_REGION
	            ELSE
	                REGION 7.3.2 - Reverse

	                    IF #ix_PEC_BoS       // Count displacement when the PE do not detects the product
	                    THEN

	                        IF #sdi_AuxGapTailtoHeadCounter_Rvs < #ci_OverflowLimit        // Prevent integer variable overflow
	                        THEN

	                            #sdi_AuxGapTailtoHeadCounter_Rvs -= #iq_UDT_ConveyorInterface.Displacement;    // Calculate the gap

	                        END_IF;
	                    END_IF;

	                END_REGION
	            END_IF;
	        END_REGION

	        REGION 7.4 - Head to head

	            // The functionality head to head is used to calculate the distance between one head's parcel and the head's parcel behind.
	            // To do it, everytime the PEC is triggered, the function save the distance calculated and reset the counter to start
	            // counting again, over and over again.
	            IF NOT #sx_ReverseDirection
	            THEN
	                REGION 7.4.1 - Forward

	                    IF #sdi_AuxGapHeadToHeadCounter_Fwd < #ci_OverflowLimit        // Prevent integer variable overflow
	                    THEN

	                        #sdi_AuxGapHeadToHeadCounter_Fwd += #iq_UDT_ConveyorInterface.Displacement;   // measure the distance between two products

	                    END_IF;

	                END_REGION
	            ELSE
	                REGION 7.4.2 - Reverse

	                    IF #sdi_AuxGapHeadToHeadCounter_Rvs < #ci_OverflowLimit        // Prevent integer variable overflow
	                    THEN

	                        #sdi_AuxGapHeadToHeadCounter_Rvs -= #iq_UDT_ConveyorInterface.Displacement;   // measure the distance between two products

	                    END_IF;

	                END_REGION
	            END_IF;
	        END_REGION

	        REGION 7.5 - Check gaps between products

	            // Check gaps is a routine that checks all the time if the gap and head to head distance is acording to the configuration.
	            // If not, the bit "sx_Gapping" is set true and the conveyor stops to gap.
	            // Compare gaps calculated with the configured gaps
	            IF NOT #sx_ReverseDirection
	            THEN
	                REGION 7.5.1 - Forward

	                    IF ((#sdi_GapHeadToHeadConfiguration_Fwd > #sdi_GapHeadToHead_Fwd               // Compare head to head configured with real distance
	                        OR #sdi_GapTailToHeadConfiguration_Fwd > #sdi_Gap_Fwd
	                        OR #sdi_GapTailToHeadConfiguration_Fwd > #sdi_DownstreamGapTailtoHead_Fwd           // Compare gap configured with real gap
	                        OR #sdi_GapHeadToHeadConfiguration_Fwd > #sdi_DownstreamGapHeadToHead_Fwd)
	                        AND #F_TRIG_AuxHeadToEnd_Fwd.Q)                                                         // Trigger when parcel arrive in the end of the conveyor
	                    THEN

	                        #sx_Gapping_Fwd := TRUE;        // Bit to inform the system that conveyor needs to stop to apply gap

	                    END_IF;

	                END_REGION
	            ELSE
	                REGION 7.5.1 - Reverse

	                    IF ((#sdi_GapHeadToHeadConfiguration_Rvs > #sdi_GapHeadToHead_Rvs               // Compare head to head configured with real distance
	                        OR #sdi_GapTailToHeadConfiguration_Rvs > #sdi_Gap_Rvs
	                        OR #sdi_GapTailToHeadConfiguration_Rvs > #sdi_DownstreamGapTailtoHead_Rvs           // Compare gap configured with real gap
	                        OR #sdi_GapHeadToHeadConfiguration_Rvs > #sdi_DownstreamGapHeadToHead_Rvs)
	                        AND #F_TRIG_AuxHeadToEnd_Rvs.Q)                                                         // Trigger when parcel arrive in the end of the conveyor
	                    THEN

	                        #sx_Gapping_Rvs := TRUE;        // Bit to inform the system that conveyor needs to stop to apply gap

	                    END_IF;

	                END_REGION
	            END_IF;
	            //    When conveyor stops to gapping, displacement values from downstream are used to
	            //    apply new gap.
	            //    When the new gap applied fits with the configured one, the conveyor starts running again.
	            //    If the conveyor stops for die back reason and the gap its been applied, and extra gap value it will be applied.
	            //    This recovery gap it helps to recovery the system after die back.
	            IF NOT #sx_ReverseDirection
	            THEN
	                REGION 7.5.3 - Forward

	                    IF (#sx_Gapping_Fwd          // Gapping needs to be applied bit
	                        AND ((#sdi_GapHeadToHeadConfiguration_Fwd > #sdi_GapHeadToHead_Fwd    // Configured head to head bigger than the actual one
	                        OR #sdi_GapHeadToHeadConfiguration_Fwd - #idi_PEC_EoSDistance / 10 + #sdi_PECtoEndDistance_Fwd > #sdi_DownstreamGapHeadToHead_Fwd
	                        OR #sdi_GapTailToHeadConfiguration_Fwd > #sdi_Gap_Fwd     // Configured gap bigger than the actual one
	                        OR #sdi_GapTailToHeadConfiguration_Fwd - #idi_PEC_EoSDistance / 10 + #sdi_PECtoEndDistance_Fwd > #sdi_DownstreamGapTailtoHead_Fwd)
	                        AND NOT #sx_RecoveryGap_Fwd)                                                // Die back recovery gap bit not active
	                        OR (((#sdi_GapHeadToHeadConfiguration_Fwd + #i_UDT_ConveyorConfiguration.ExtraGapRecovery)   // Add recovery gap to the configured
	                        > #sdi_GapHeadToHead_Fwd                                                                                 // Actual head to head distance
	                        OR (#sdi_GapHeadToHeadConfiguration_Fwd - #idi_PEC_EoSDistance / 10 + #sdi_PECtoEndDistance_Fwd + #i_UDT_ConveyorConfiguration.ExtraGapRecovery)
	                        > #sdi_DownstreamGapHeadToHead_Fwd
	                        OR (#sdi_GapTailToHeadConfiguration_Fwd + #i_UDT_ConveyorConfiguration.ExtraGapRecovery)    // Add recovery gap to the configured
	                        > #sdi_Gap_Fwd                                                                               // Actual gap between parcels
	                        OR (#sdi_GapTailToHeadConfiguration_Fwd - #idi_PEC_EoSDistance / 10 + #sdi_PECtoEndDistance_Fwd + #i_UDT_ConveyorConfiguration.ExtraGapRecovery)
	                        > #sdi_DownstreamGapTailtoHead_Fwd)
	                        AND #sx_RecoveryGap_Fwd))                                                                       // Recovery gap bit activate
	                    THEN

	                        #sdi_GapHeadToHead_Fwd += #iq_UDT_HandShake.DownstreamDisplacement;      // Increase head to head counter with conveyor downstream displacement
	                        #sdi_Gap_Fwd += #iq_UDT_HandShake.DownstreamDisplacement;     // Increase gap counter with conveyor downstream displacement

	                    ELSE

	                        #sx_Gapping_Fwd := FALSE;                   // Set gapping bit to false

	                    END_IF;

	                    IF #sx_Gapping_Fwd                              // Gapping bit active
	                        AND NOT #iq_UDT_HandShake.RTR           // Ready to receive not active
	                    THEN

	                        #sx_RecoveryGap_Fwd := TRUE;                // Recovery gap activation after die back

	                    END_IF;

	                    IF #sx_RecoveryGap_Fwd                          // Recovery gap active
	                        AND NOT #sx_Gapping_Fwd                     // Gapping bit not active
	                    THEN

	                        #sx_RecoveryGap_Fwd := FALSE;               // Recovery gap disable

	                    END_IF;

	                END_REGION
	            ELSE
	                REGION 7.5.4 - Reverse

